// TIA Portal V17 export
// export: Created 2025-03-07T09:19:12.8663943Z, ExportSetting WithDefaults, DisplayName Totally Integrated Automation Portal, DisplayVersion V17 Update 8, DisplayName TIA Portal Openness, DisplayVersion V17 Update 8, DisplayName TIA Portal Version Control Interface, DisplayVersion V17, DisplayName SINAMICS Startdrive Advanced, DisplayVersion V17 SP2, DisplayName SINAMICS Startdrive G110M, G120, G120C, G120D, G120P, G115D, DisplayVersion V17 SP2, DisplayName SINAMICS Startdrive G130, G150, S120, S150, SINAMICS MV, S210, DisplayVersion V17 SP2, DisplayName STEP 7 Professional, DisplayVersion V17 Update 8, DisplayName SINUMERIK ONE STEP 7 Toolbox, DisplayVersion V17 Update 12, DisplayName SINUMERIK 840D sl STEP 7 Toolbox, DisplayVersion V17 Update 12, DisplayName STEP 7 Safety, DisplayVersion V17 Update 6, DisplayName WinCC Advanced, DisplayVersion V17 Update 8
FUNCTION "FC7236_SHOW_HIDE_ELEMENTS_CLADDING" : Void   // FC7236, LAD
{ S7_Optimized_Access := 'FALSE' }
AUTHOR : ETXETAR
VERSION : 1.0
// stored: AutoNumber false, IsIECCheckEnabled false, SetENOAutomatically false, UDAEnableTagReadback false
   VAR_TEMP
      ONE : Byte;
      RETVAL_FILL : Int;
      ZERO : Byte;
      MINUS_ONE : Byte;
      SHOW_TABLES : Bool;
      NO_REASON_CODE : Bool;
      AXIS_AUX1 : Bool;
      AXIS_AUX2 : Bool;
   END_VAR
   VAR_TEMP   // added for the SCL form of the ladder/FBD networks
      _w1 : Bool;
      _w2 : Bool;
   END_VAR
BEGIN

REGION Network 1: MOVE VALUES
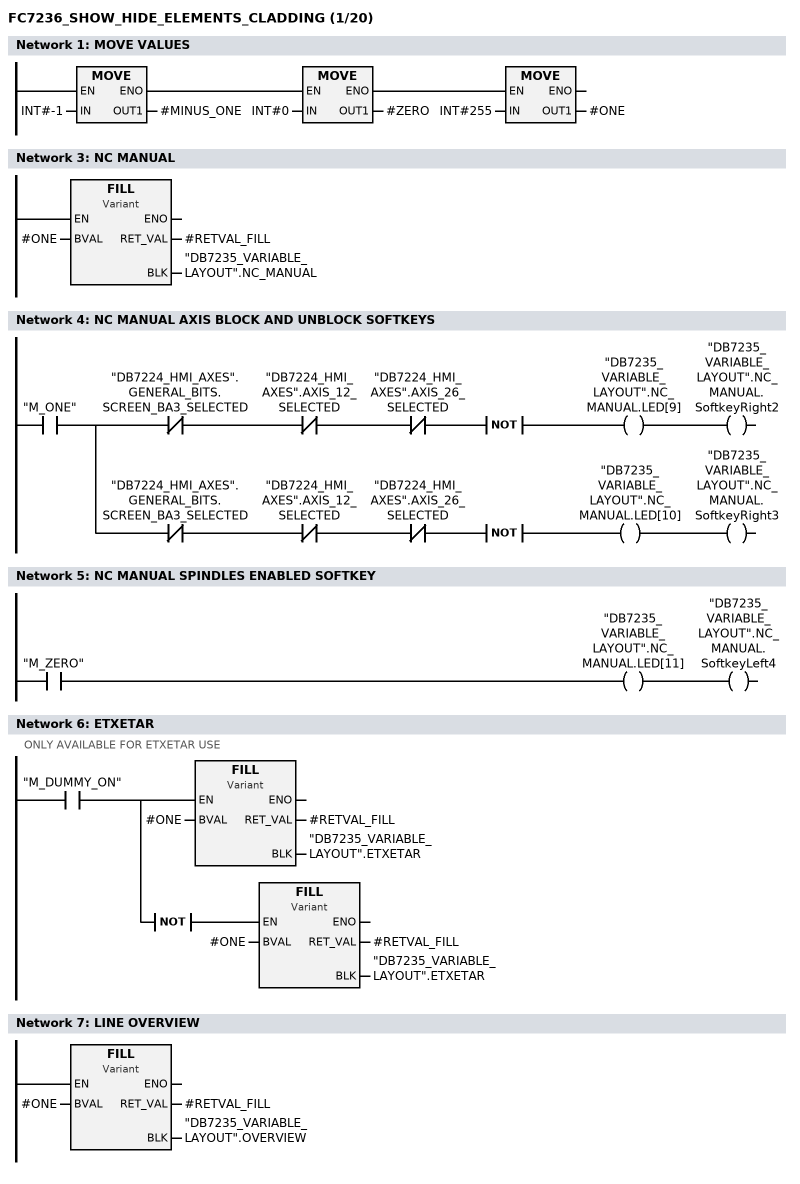
   RUNG wire#powerrail
      { S7_GenerateENO := "TRUE" } Move(in := INT#-1, out1 => #MINUS_ONE)
      { S7_GenerateENO := "TRUE" } Move(in := INT#0, out1 => #ZERO)
      { S7_GenerateENO := "TRUE" } Move(in := INT#255, out1 => #ONE)
   END_RUNG
   // the same network as SCL:
   // ENO of a box is taken as its EN; it also drops when the box reports an error
   #MINUS_ONE := INT#-1;
   #ZERO := INT#0;
   #ONE := INT#255;
END_REGION

REGION Network 2: *************** SHOW OR HIDE ELEMENTS ***************
END_REGION

REGION Network 3: NC MANUAL
   RUNG wire#powerrail
      { S7_Templates := "ptr_type := Variant" } FILL(BVAL := #ONE, RET_VAL => #RETVAL_FILL, BLK => "DB7235_VARIABLE_LAYOUT".NC_MANUAL)
   END_RUNG
   // the same network as SCL:
   #RETVAL_FILL := FILL(BVAL := #ONE, BLK => "DB7235_VARIABLE_LAYOUT".NC_MANUAL);
END_REGION

REGION Network 4: NC MANUAL AXIS BLOCK AND UNBLOCK SOFTKEYS
   RUNG wire#powerrail
      Contact( "M_ONE" )
      wire#w1
      I_Contact( "DB7224_HMI_AXES".GENERAL_BITS.SCREEN_BA3_SELECTED )
      I_Contact( "DB7224_HMI_AXES".AXIS_12_SELECTED )
      I_Contact( "DB7224_HMI_AXES".AXIS_26_SELECTED )
      Not()
      Coil( "DB7235_VARIABLE_LAYOUT".NC_MANUAL.LED[9] )
      Coil( "DB7235_VARIABLE_LAYOUT".NC_MANUAL.SoftkeyRight2 )
   END_RUNG
   RUNG wire#w1
      I_Contact( "DB7224_HMI_AXES".GENERAL_BITS.SCREEN_BA3_SELECTED )
      I_Contact( "DB7224_HMI_AXES".AXIS_12_SELECTED )
      I_Contact( "DB7224_HMI_AXES".AXIS_26_SELECTED )
      Not()
      Coil( "DB7235_VARIABLE_LAYOUT".NC_MANUAL.LED[10] )
      Coil( "DB7235_VARIABLE_LAYOUT".NC_MANUAL.SoftkeyRight3 )
   END_RUNG
   // the same network as SCL:
   "DB7235_VARIABLE_LAYOUT".NC_MANUAL.LED[9] := NOT ("M_ONE" AND NOT "DB7224_HMI_AXES".GENERAL_BITS.SCREEN_BA3_SELECTED AND NOT "DB7224_HMI_AXES".AXIS_12_SELECTED AND NOT "DB7224_HMI_AXES".AXIS_26_SELECTED);
   "DB7235_VARIABLE_LAYOUT".NC_MANUAL.SoftkeyRight2 := NOT ("M_ONE" AND NOT "DB7224_HMI_AXES".GENERAL_BITS.SCREEN_BA3_SELECTED AND NOT "DB7224_HMI_AXES".AXIS_12_SELECTED AND NOT "DB7224_HMI_AXES".AXIS_26_SELECTED);
   "DB7235_VARIABLE_LAYOUT".NC_MANUAL.LED[10] := NOT ("M_ONE" AND NOT "DB7224_HMI_AXES".GENERAL_BITS.SCREEN_BA3_SELECTED AND NOT "DB7224_HMI_AXES".AXIS_12_SELECTED AND NOT "DB7224_HMI_AXES".AXIS_26_SELECTED);
   "DB7235_VARIABLE_LAYOUT".NC_MANUAL.SoftkeyRight3 := NOT ("M_ONE" AND NOT "DB7224_HMI_AXES".GENERAL_BITS.SCREEN_BA3_SELECTED AND NOT "DB7224_HMI_AXES".AXIS_12_SELECTED AND NOT "DB7224_HMI_AXES".AXIS_26_SELECTED);
END_REGION

REGION Network 5: NC MANUAL SPINDLES ENABLED SOFTKEY
   RUNG wire#powerrail
      Contact( "M_ZERO" )
      Coil( "DB7235_VARIABLE_LAYOUT".NC_MANUAL.LED[11] )
      Coil( "DB7235_VARIABLE_LAYOUT".NC_MANUAL.SoftkeyLeft4 )
   END_RUNG
   // the same network as SCL:
   "DB7235_VARIABLE_LAYOUT".NC_MANUAL.LED[11] := "M_ZERO";
   "DB7235_VARIABLE_LAYOUT".NC_MANUAL.SoftkeyLeft4 := "M_ZERO";
END_REGION

REGION Network 6: ETXETAR
   // ONLY AVAILABLE FOR ETXETAR USE
   RUNG wire#powerrail
      Contact( "M_DUMMY_ON" )
      wire#w1
      { S7_Templates := "ptr_type := Variant" } FILL(BVAL := #ONE, RET_VAL => #RETVAL_FILL, BLK => "DB7235_VARIABLE_LAYOUT".ETXETAR)
   END_RUNG
   RUNG wire#w1
      Not()
      { S7_Templates := "ptr_type := Variant" } FILL(BVAL := #ONE, RET_VAL => #RETVAL_FILL, BLK => "DB7235_VARIABLE_LAYOUT".ETXETAR)
   END_RUNG
   // the same network as SCL:
   #_w1 := "M_DUMMY_ON";
   IF #_w1 THEN #RETVAL_FILL := FILL(BVAL := #ONE, BLK => "DB7235_VARIABLE_LAYOUT".ETXETAR); END_IF;
   IF NOT #_w1 THEN #RETVAL_FILL := FILL(BVAL := #ONE, BLK => "DB7235_VARIABLE_LAYOUT".ETXETAR); END_IF;
END_REGION

REGION Network 7: LINE OVERVIEW
   RUNG wire#powerrail
      { S7_Templates := "ptr_type := Variant" } FILL(BVAL := #ONE, RET_VAL => #RETVAL_FILL, BLK => "DB7235_VARIABLE_LAYOUT".OVERVIEW)
   END_RUNG
   // the same network as SCL:
   #RETVAL_FILL := FILL(BVAL := #ONE, BLK => "DB7235_VARIABLE_LAYOUT".OVERVIEW);
END_REGION

REGION Network 8: LINE OVERVIEW IO FIELD AND TEXTS
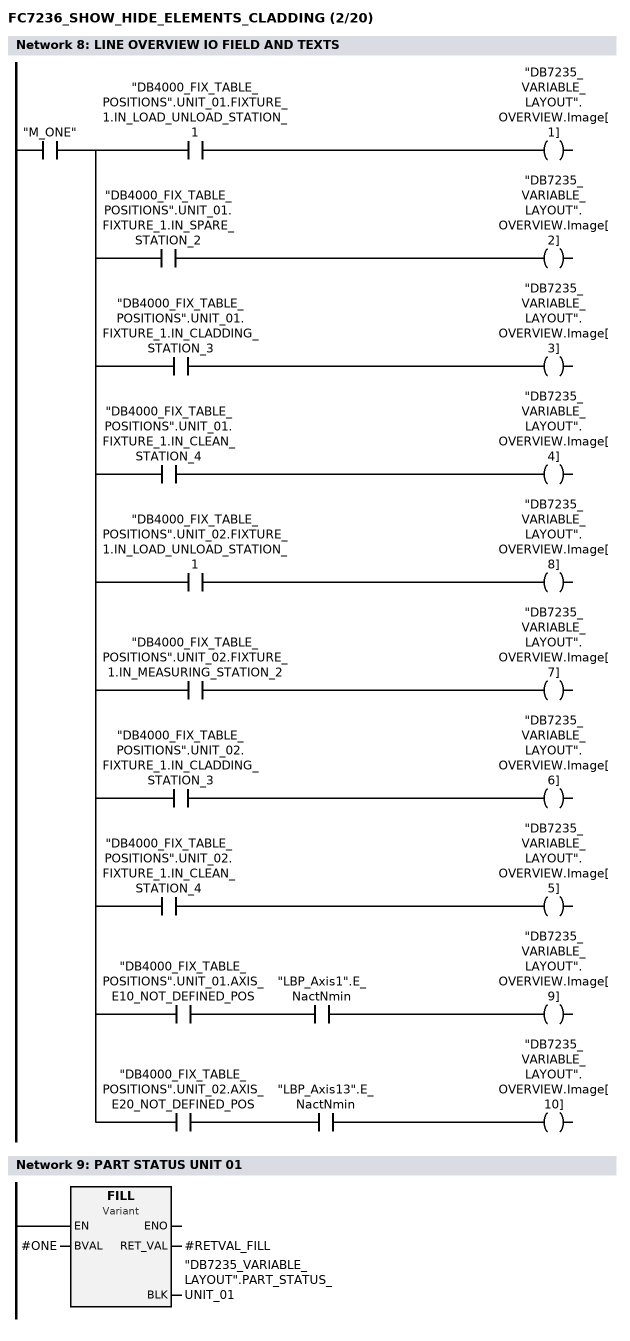
   RUNG wire#powerrail
      Contact( "M_ONE" )
      wire#w1
      Contact( "DB4000_FIX_TABLE_POSITIONS".UNIT_01.FIXTURE_1.IN_LOAD_UNLOAD_STATION_1 )
      Coil( "DB7235_VARIABLE_LAYOUT".OVERVIEW.Image[1] )
   END_RUNG
   RUNG wire#w1
      Contact( "DB4000_FIX_TABLE_POSITIONS".UNIT_01.FIXTURE_1.IN_SPARE_STATION_2 )
      Coil( "DB7235_VARIABLE_LAYOUT".OVERVIEW.Image[2] )
   END_RUNG
   RUNG wire#w1
      Contact( "DB4000_FIX_TABLE_POSITIONS".UNIT_01.FIXTURE_1.IN_CLADDING_STATION_3 )
      Coil( "DB7235_VARIABLE_LAYOUT".OVERVIEW.Image[3] )
   END_RUNG
   RUNG wire#w1
      Contact( "DB4000_FIX_TABLE_POSITIONS".UNIT_01.FIXTURE_1.IN_CLEAN_STATION_4 )
      Coil( "DB7235_VARIABLE_LAYOUT".OVERVIEW.Image[4] )
   END_RUNG
   RUNG wire#w1
      Contact( "DB4000_FIX_TABLE_POSITIONS".UNIT_02.FIXTURE_1.IN_LOAD_UNLOAD_STATION_1 )
      Coil( "DB7235_VARIABLE_LAYOUT".OVERVIEW.Image[8] )
   END_RUNG
   RUNG wire#w1
      Contact( "DB4000_FIX_TABLE_POSITIONS".UNIT_02.FIXTURE_1.IN_MEASURING_STATION_2 )
      Coil( "DB7235_VARIABLE_LAYOUT".OVERVIEW.Image[7] )
   END_RUNG
   RUNG wire#w1
      Contact( "DB4000_FIX_TABLE_POSITIONS".UNIT_02.FIXTURE_1.IN_CLADDING_STATION_3 )
      Coil( "DB7235_VARIABLE_LAYOUT".OVERVIEW.Image[6] )
   END_RUNG
   RUNG wire#w1
      Contact( "DB4000_FIX_TABLE_POSITIONS".UNIT_02.FIXTURE_1.IN_CLEAN_STATION_4 )
      Coil( "DB7235_VARIABLE_LAYOUT".OVERVIEW.Image[5] )
   END_RUNG
   RUNG wire#w1
      Contact( "DB4000_FIX_TABLE_POSITIONS".UNIT_01.AXIS_E10_NOT_DEFINED_POS )
      Contact( "LBP_Axis1".E_NactNmin )
      Coil( "DB7235_VARIABLE_LAYOUT".OVERVIEW.Image[9] )
   END_RUNG
   RUNG wire#w1
      Contact( "DB4000_FIX_TABLE_POSITIONS".UNIT_02.AXIS_E20_NOT_DEFINED_POS )
      Contact( "LBP_Axis13".E_NactNmin )
      Coil( "DB7235_VARIABLE_LAYOUT".OVERVIEW.Image[10] )
   END_RUNG
   // the same network as SCL:
   "DB7235_VARIABLE_LAYOUT".OVERVIEW.Image[1] := "M_ONE" AND "DB4000_FIX_TABLE_POSITIONS".UNIT_01.FIXTURE_1.IN_LOAD_UNLOAD_STATION_1;
   "DB7235_VARIABLE_LAYOUT".OVERVIEW.Image[2] := "M_ONE" AND "DB4000_FIX_TABLE_POSITIONS".UNIT_01.FIXTURE_1.IN_SPARE_STATION_2;
   "DB7235_VARIABLE_LAYOUT".OVERVIEW.Image[3] := "M_ONE" AND "DB4000_FIX_TABLE_POSITIONS".UNIT_01.FIXTURE_1.IN_CLADDING_STATION_3;
   "DB7235_VARIABLE_LAYOUT".OVERVIEW.Image[4] := "M_ONE" AND "DB4000_FIX_TABLE_POSITIONS".UNIT_01.FIXTURE_1.IN_CLEAN_STATION_4;
   "DB7235_VARIABLE_LAYOUT".OVERVIEW.Image[8] := "M_ONE" AND "DB4000_FIX_TABLE_POSITIONS".UNIT_02.FIXTURE_1.IN_LOAD_UNLOAD_STATION_1;
   "DB7235_VARIABLE_LAYOUT".OVERVIEW.Image[7] := "M_ONE" AND "DB4000_FIX_TABLE_POSITIONS".UNIT_02.FIXTURE_1.IN_MEASURING_STATION_2;
   "DB7235_VARIABLE_LAYOUT".OVERVIEW.Image[6] := "M_ONE" AND "DB4000_FIX_TABLE_POSITIONS".UNIT_02.FIXTURE_1.IN_CLADDING_STATION_3;
   "DB7235_VARIABLE_LAYOUT".OVERVIEW.Image[5] := "M_ONE" AND "DB4000_FIX_TABLE_POSITIONS".UNIT_02.FIXTURE_1.IN_CLEAN_STATION_4;
   "DB7235_VARIABLE_LAYOUT".OVERVIEW.Image[9] := "M_ONE" AND "DB4000_FIX_TABLE_POSITIONS".UNIT_01.AXIS_E10_NOT_DEFINED_POS AND "LBP_Axis1".E_NactNmin;
   "DB7235_VARIABLE_LAYOUT".OVERVIEW.Image[10] := "M_ONE" AND "DB4000_FIX_TABLE_POSITIONS".UNIT_02.AXIS_E20_NOT_DEFINED_POS AND "LBP_Axis13".E_NactNmin;
END_REGION

REGION Network 9: PART STATUS UNIT 01
   RUNG wire#powerrail
      { S7_Templates := "ptr_type := Variant" } FILL(BVAL := #ONE, RET_VAL => #RETVAL_FILL, BLK => "DB7235_VARIABLE_LAYOUT".PART_STATUS_UNIT_01)
   END_RUNG
   // the same network as SCL:
   #RETVAL_FILL := FILL(BVAL := #ONE, BLK => "DB7235_VARIABLE_LAYOUT".PART_STATUS_UNIT_01);
END_REGION

REGION Network 10: PART STATUS IO FIELD AND TEXTS UNIT 01
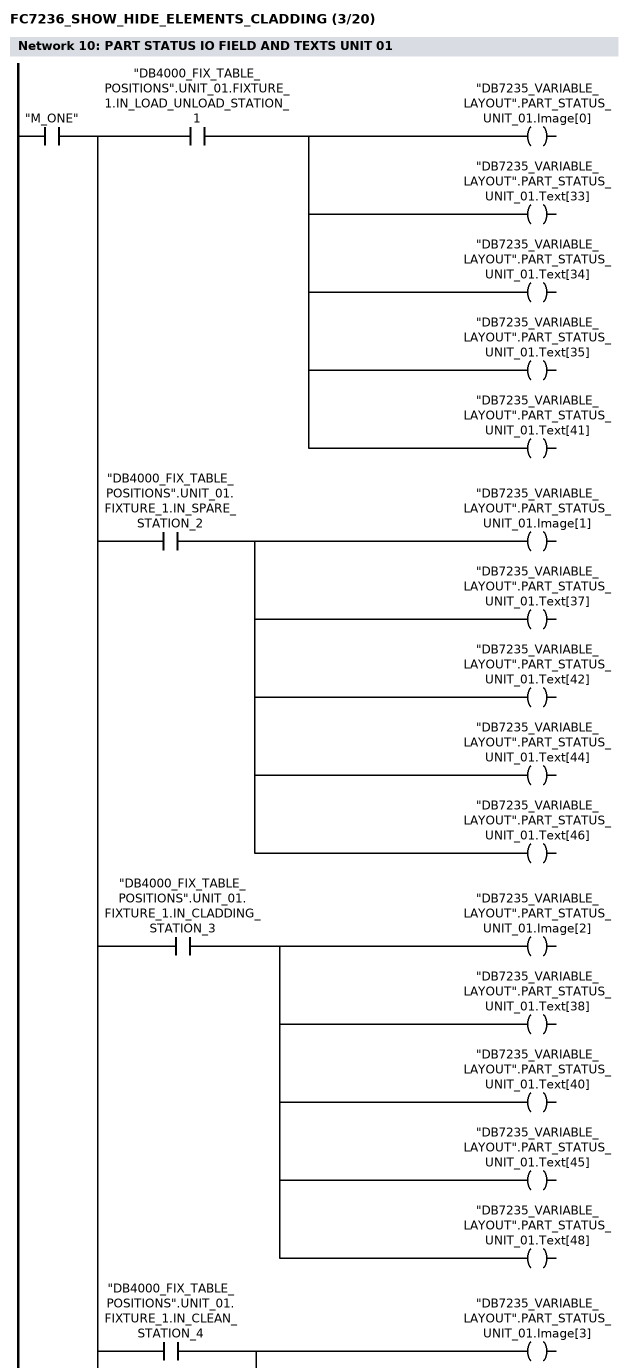
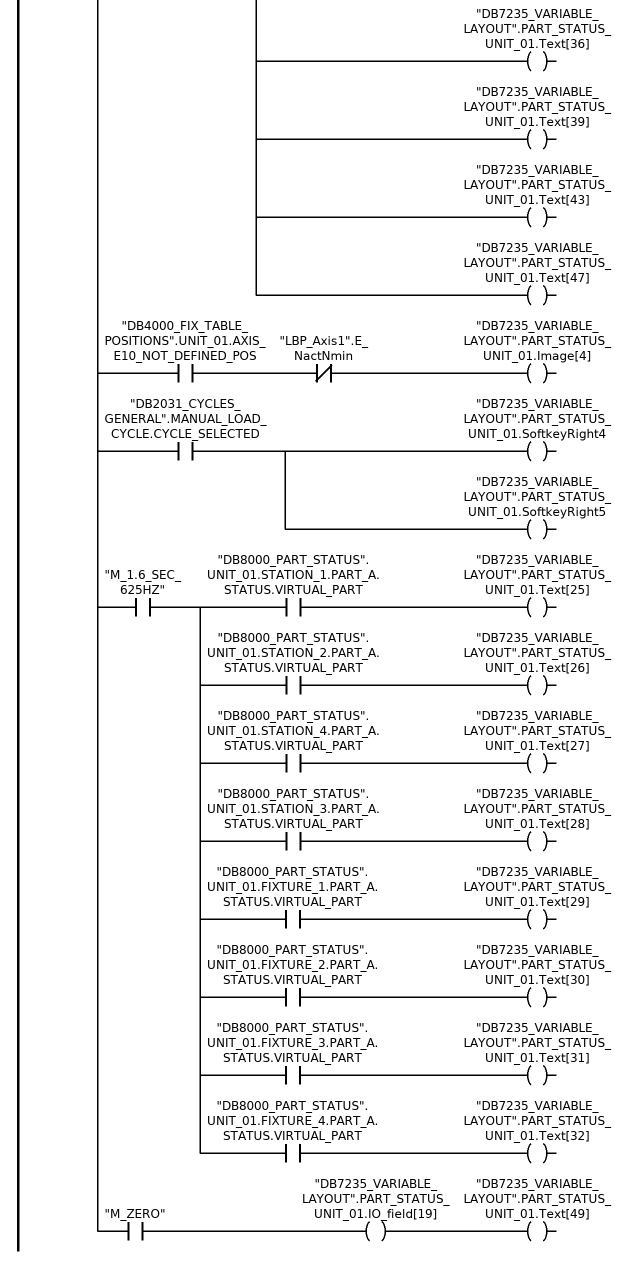
   RUNG wire#powerrail
      Contact( "M_ONE" )
      wire#w1
      Contact( "DB4000_FIX_TABLE_POSITIONS".UNIT_01.FIXTURE_1.IN_LOAD_UNLOAD_STATION_1 )
      wire#w2
      Coil( "DB7235_VARIABLE_LAYOUT".PART_STATUS_UNIT_01.Image[0] )
   END_RUNG
   RUNG wire#w2
      Coil( "DB7235_VARIABLE_LAYOUT".PART_STATUS_UNIT_01.Text[33] )
   END_RUNG
   RUNG wire#w2
      Coil( "DB7235_VARIABLE_LAYOUT".PART_STATUS_UNIT_01.Text[34] )
   END_RUNG
   RUNG wire#w2
      Coil( "DB7235_VARIABLE_LAYOUT".PART_STATUS_UNIT_01.Text[35] )
   END_RUNG
   RUNG wire#w2
      Coil( "DB7235_VARIABLE_LAYOUT".PART_STATUS_UNIT_01.Text[41] )
   END_RUNG
   RUNG wire#w1
      Contact( "DB4000_FIX_TABLE_POSITIONS".UNIT_01.FIXTURE_1.IN_SPARE_STATION_2 )
      wire#w3
      Coil( "DB7235_VARIABLE_LAYOUT".PART_STATUS_UNIT_01.Image[1] )
   END_RUNG
   RUNG wire#w3
      Coil( "DB7235_VARIABLE_LAYOUT".PART_STATUS_UNIT_01.Text[37] )
   END_RUNG
   RUNG wire#w3
      Coil( "DB7235_VARIABLE_LAYOUT".PART_STATUS_UNIT_01.Text[42] )
   END_RUNG
   RUNG wire#w3
      Coil( "DB7235_VARIABLE_LAYOUT".PART_STATUS_UNIT_01.Text[44] )
   END_RUNG
   RUNG wire#w3
      Coil( "DB7235_VARIABLE_LAYOUT".PART_STATUS_UNIT_01.Text[46] )
   END_RUNG
   RUNG wire#w1
      Contact( "DB4000_FIX_TABLE_POSITIONS".UNIT_01.FIXTURE_1.IN_CLADDING_STATION_3 )
      wire#w4
      Coil( "DB7235_VARIABLE_LAYOUT".PART_STATUS_UNIT_01.Image[2] )
   END_RUNG
   RUNG wire#w4
      Coil( "DB7235_VARIABLE_LAYOUT".PART_STATUS_UNIT_01.Text[38] )
   END_RUNG
   RUNG wire#w4
      Coil( "DB7235_VARIABLE_LAYOUT".PART_STATUS_UNIT_01.Text[40] )
   END_RUNG
   RUNG wire#w4
      Coil( "DB7235_VARIABLE_LAYOUT".PART_STATUS_UNIT_01.Text[45] )
   END_RUNG
   RUNG wire#w4
      Coil( "DB7235_VARIABLE_LAYOUT".PART_STATUS_UNIT_01.Text[48] )
   END_RUNG
   RUNG wire#w1
      Contact( "DB4000_FIX_TABLE_POSITIONS".UNIT_01.FIXTURE_1.IN_CLEAN_STATION_4 )
      wire#w5
      Coil( "DB7235_VARIABLE_LAYOUT".PART_STATUS_UNIT_01.Image[3] )
   END_RUNG
   RUNG wire#w5
      Coil( "DB7235_VARIABLE_LAYOUT".PART_STATUS_UNIT_01.Text[36] )
   END_RUNG
   RUNG wire#w5
      Coil( "DB7235_VARIABLE_LAYOUT".PART_STATUS_UNIT_01.Text[39] )
   END_RUNG
   RUNG wire#w5
      Coil( "DB7235_VARIABLE_LAYOUT".PART_STATUS_UNIT_01.Text[43] )
   END_RUNG
   RUNG wire#w5
      Coil( "DB7235_VARIABLE_LAYOUT".PART_STATUS_UNIT_01.Text[47] )
   END_RUNG
   RUNG wire#w1
      Contact( "DB4000_FIX_TABLE_POSITIONS".UNIT_01.AXIS_E10_NOT_DEFINED_POS )
      I_Contact( "LBP_Axis1".E_NactNmin )
      Coil( "DB7235_VARIABLE_LAYOUT".PART_STATUS_UNIT_01.Image[4] )
   END_RUNG
   RUNG wire#w1
      Contact( "DB2031_CYCLES_GENERAL".MANUAL_LOAD_CYCLE.CYCLE_SELECTED )
      wire#w6
      Coil( "DB7235_VARIABLE_LAYOUT".PART_STATUS_UNIT_01.SoftkeyRight4 )
   END_RUNG
   RUNG wire#w6
      Coil( "DB7235_VARIABLE_LAYOUT".PART_STATUS_UNIT_01.SoftkeyRight5 )
   END_RUNG
   RUNG wire#w1
      Contact( "M_1.6_SEC_625HZ" )
      wire#w7
      Contact( "DB8000_PART_STATUS".UNIT_01.STATION_1.PART_A.STATUS.VIRTUAL_PART )
      Coil( "DB7235_VARIABLE_LAYOUT".PART_STATUS_UNIT_01.Text[25] )
   END_RUNG
   RUNG wire#w7
      Contact( "DB8000_PART_STATUS".UNIT_01.STATION_2.PART_A.STATUS.VIRTUAL_PART )
      Coil( "DB7235_VARIABLE_LAYOUT".PART_STATUS_UNIT_01.Text[26] )
   END_RUNG
   RUNG wire#w7
      Contact( "DB8000_PART_STATUS".UNIT_01.STATION_4.PART_A.STATUS.VIRTUAL_PART )
      Coil( "DB7235_VARIABLE_LAYOUT".PART_STATUS_UNIT_01.Text[27] )
   END_RUNG
   RUNG wire#w7
      Contact( "DB8000_PART_STATUS".UNIT_01.STATION_3.PART_A.STATUS.VIRTUAL_PART )
      Coil( "DB7235_VARIABLE_LAYOUT".PART_STATUS_UNIT_01.Text[28] )
   END_RUNG
   RUNG wire#w7
      Contact( "DB8000_PART_STATUS".UNIT_01.FIXTURE_1.PART_A.STATUS.VIRTUAL_PART )
      Coil( "DB7235_VARIABLE_LAYOUT".PART_STATUS_UNIT_01.Text[29] )
   END_RUNG
   RUNG wire#w7
      Contact( "DB8000_PART_STATUS".UNIT_01.FIXTURE_2.PART_A.STATUS.VIRTUAL_PART )
      Coil( "DB7235_VARIABLE_LAYOUT".PART_STATUS_UNIT_01.Text[30] )
   END_RUNG
   RUNG wire#w7
      Contact( "DB8000_PART_STATUS".UNIT_01.FIXTURE_3.PART_A.STATUS.VIRTUAL_PART )
      Coil( "DB7235_VARIABLE_LAYOUT".PART_STATUS_UNIT_01.Text[31] )
   END_RUNG
   RUNG wire#w7
      Contact( "DB8000_PART_STATUS".UNIT_01.FIXTURE_4.PART_A.STATUS.VIRTUAL_PART )
      Coil( "DB7235_VARIABLE_LAYOUT".PART_STATUS_UNIT_01.Text[32] )
   END_RUNG
   RUNG wire#w1
      Contact( "M_ZERO" )
      Coil( "DB7235_VARIABLE_LAYOUT".PART_STATUS_UNIT_01.IO_field[19] )
      Coil( "DB7235_VARIABLE_LAYOUT".PART_STATUS_UNIT_01.Text[49] )
   END_RUNG
   // the same network as SCL:
   "DB7235_VARIABLE_LAYOUT".PART_STATUS_UNIT_01.Image[0] := "M_ONE" AND "DB4000_FIX_TABLE_POSITIONS".UNIT_01.FIXTURE_1.IN_LOAD_UNLOAD_STATION_1;
   "DB7235_VARIABLE_LAYOUT".PART_STATUS_UNIT_01.Text[33] := "M_ONE" AND "DB4000_FIX_TABLE_POSITIONS".UNIT_01.FIXTURE_1.IN_LOAD_UNLOAD_STATION_1;
   "DB7235_VARIABLE_LAYOUT".PART_STATUS_UNIT_01.Text[34] := "M_ONE" AND "DB4000_FIX_TABLE_POSITIONS".UNIT_01.FIXTURE_1.IN_LOAD_UNLOAD_STATION_1;
   "DB7235_VARIABLE_LAYOUT".PART_STATUS_UNIT_01.Text[35] := "M_ONE" AND "DB4000_FIX_TABLE_POSITIONS".UNIT_01.FIXTURE_1.IN_LOAD_UNLOAD_STATION_1;
   "DB7235_VARIABLE_LAYOUT".PART_STATUS_UNIT_01.Text[41] := "M_ONE" AND "DB4000_FIX_TABLE_POSITIONS".UNIT_01.FIXTURE_1.IN_LOAD_UNLOAD_STATION_1;
   "DB7235_VARIABLE_LAYOUT".PART_STATUS_UNIT_01.Image[1] := "M_ONE" AND "DB4000_FIX_TABLE_POSITIONS".UNIT_01.FIXTURE_1.IN_SPARE_STATION_2;
   "DB7235_VARIABLE_LAYOUT".PART_STATUS_UNIT_01.Text[37] := "M_ONE" AND "DB4000_FIX_TABLE_POSITIONS".UNIT_01.FIXTURE_1.IN_SPARE_STATION_2;
   "DB7235_VARIABLE_LAYOUT".PART_STATUS_UNIT_01.Text[42] := "M_ONE" AND "DB4000_FIX_TABLE_POSITIONS".UNIT_01.FIXTURE_1.IN_SPARE_STATION_2;
   "DB7235_VARIABLE_LAYOUT".PART_STATUS_UNIT_01.Text[44] := "M_ONE" AND "DB4000_FIX_TABLE_POSITIONS".UNIT_01.FIXTURE_1.IN_SPARE_STATION_2;
   "DB7235_VARIABLE_LAYOUT".PART_STATUS_UNIT_01.Text[46] := "M_ONE" AND "DB4000_FIX_TABLE_POSITIONS".UNIT_01.FIXTURE_1.IN_SPARE_STATION_2;
   "DB7235_VARIABLE_LAYOUT".PART_STATUS_UNIT_01.Image[2] := "M_ONE" AND "DB4000_FIX_TABLE_POSITIONS".UNIT_01.FIXTURE_1.IN_CLADDING_STATION_3;
   "DB7235_VARIABLE_LAYOUT".PART_STATUS_UNIT_01.Text[38] := "M_ONE" AND "DB4000_FIX_TABLE_POSITIONS".UNIT_01.FIXTURE_1.IN_CLADDING_STATION_3;
   "DB7235_VARIABLE_LAYOUT".PART_STATUS_UNIT_01.Text[40] := "M_ONE" AND "DB4000_FIX_TABLE_POSITIONS".UNIT_01.FIXTURE_1.IN_CLADDING_STATION_3;
   "DB7235_VARIABLE_LAYOUT".PART_STATUS_UNIT_01.Text[45] := "M_ONE" AND "DB4000_FIX_TABLE_POSITIONS".UNIT_01.FIXTURE_1.IN_CLADDING_STATION_3;
   "DB7235_VARIABLE_LAYOUT".PART_STATUS_UNIT_01.Text[48] := "M_ONE" AND "DB4000_FIX_TABLE_POSITIONS".UNIT_01.FIXTURE_1.IN_CLADDING_STATION_3;
   "DB7235_VARIABLE_LAYOUT".PART_STATUS_UNIT_01.Image[3] := "M_ONE" AND "DB4000_FIX_TABLE_POSITIONS".UNIT_01.FIXTURE_1.IN_CLEAN_STATION_4;
   "DB7235_VARIABLE_LAYOUT".PART_STATUS_UNIT_01.Text[36] := "M_ONE" AND "DB4000_FIX_TABLE_POSITIONS".UNIT_01.FIXTURE_1.IN_CLEAN_STATION_4;
   "DB7235_VARIABLE_LAYOUT".PART_STATUS_UNIT_01.Text[39] := "M_ONE" AND "DB4000_FIX_TABLE_POSITIONS".UNIT_01.FIXTURE_1.IN_CLEAN_STATION_4;
   "DB7235_VARIABLE_LAYOUT".PART_STATUS_UNIT_01.Text[43] := "M_ONE" AND "DB4000_FIX_TABLE_POSITIONS".UNIT_01.FIXTURE_1.IN_CLEAN_STATION_4;
   "DB7235_VARIABLE_LAYOUT".PART_STATUS_UNIT_01.Text[47] := "M_ONE" AND "DB4000_FIX_TABLE_POSITIONS".UNIT_01.FIXTURE_1.IN_CLEAN_STATION_4;
   "DB7235_VARIABLE_LAYOUT".PART_STATUS_UNIT_01.Image[4] := "M_ONE" AND "DB4000_FIX_TABLE_POSITIONS".UNIT_01.AXIS_E10_NOT_DEFINED_POS AND NOT "LBP_Axis1".E_NactNmin;
   "DB7235_VARIABLE_LAYOUT".PART_STATUS_UNIT_01.SoftkeyRight4 := "M_ONE" AND "DB2031_CYCLES_GENERAL".MANUAL_LOAD_CYCLE.CYCLE_SELECTED;
   "DB7235_VARIABLE_LAYOUT".PART_STATUS_UNIT_01.SoftkeyRight5 := "DB7235_VARIABLE_LAYOUT".PART_STATUS_UNIT_01.SoftkeyRight4;
   #_w1 := "M_ONE" AND "M_1.6_SEC_625HZ";
   "DB7235_VARIABLE_LAYOUT".PART_STATUS_UNIT_01.Text[25] := #_w1 AND "DB8000_PART_STATUS".UNIT_01.STATION_1.PART_A.STATUS.VIRTUAL_PART;
   "DB7235_VARIABLE_LAYOUT".PART_STATUS_UNIT_01.Text[26] := #_w1 AND "DB8000_PART_STATUS".UNIT_01.STATION_2.PART_A.STATUS.VIRTUAL_PART;
   "DB7235_VARIABLE_LAYOUT".PART_STATUS_UNIT_01.Text[27] := #_w1 AND "DB8000_PART_STATUS".UNIT_01.STATION_4.PART_A.STATUS.VIRTUAL_PART;
   "DB7235_VARIABLE_LAYOUT".PART_STATUS_UNIT_01.Text[28] := #_w1 AND "DB8000_PART_STATUS".UNIT_01.STATION_3.PART_A.STATUS.VIRTUAL_PART;
   "DB7235_VARIABLE_LAYOUT".PART_STATUS_UNIT_01.Text[29] := #_w1 AND "DB8000_PART_STATUS".UNIT_01.FIXTURE_1.PART_A.STATUS.VIRTUAL_PART;
   "DB7235_VARIABLE_LAYOUT".PART_STATUS_UNIT_01.Text[30] := #_w1 AND "DB8000_PART_STATUS".UNIT_01.FIXTURE_2.PART_A.STATUS.VIRTUAL_PART;
   "DB7235_VARIABLE_LAYOUT".PART_STATUS_UNIT_01.Text[31] := #_w1 AND "DB8000_PART_STATUS".UNIT_01.FIXTURE_3.PART_A.STATUS.VIRTUAL_PART;
   "DB7235_VARIABLE_LAYOUT".PART_STATUS_UNIT_01.Text[32] := #_w1 AND "DB8000_PART_STATUS".UNIT_01.FIXTURE_4.PART_A.STATUS.VIRTUAL_PART;
   "DB7235_VARIABLE_LAYOUT".PART_STATUS_UNIT_01.IO_field[19] := "M_ONE" AND "M_ZERO";
   "DB7235_VARIABLE_LAYOUT".PART_STATUS_UNIT_01.Text[49] := "M_ONE" AND "M_ZERO";
END_REGION

REGION Network 11: QUALITY CHECK
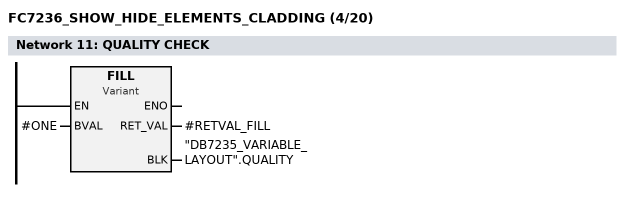
   RUNG wire#powerrail
      { S7_Templates := "ptr_type := Variant" } FILL(BVAL := #ONE, RET_VAL => #RETVAL_FILL, BLK => "DB7235_VARIABLE_LAYOUT".QUALITY)
   END_RUNG
   // the same network as SCL:
   #RETVAL_FILL := FILL(BVAL := #ONE, BLK => "DB7235_VARIABLE_LAYOUT".QUALITY);
END_REGION

REGION Network 12: QUALITY CHECK IO FIELD AND TEXTS
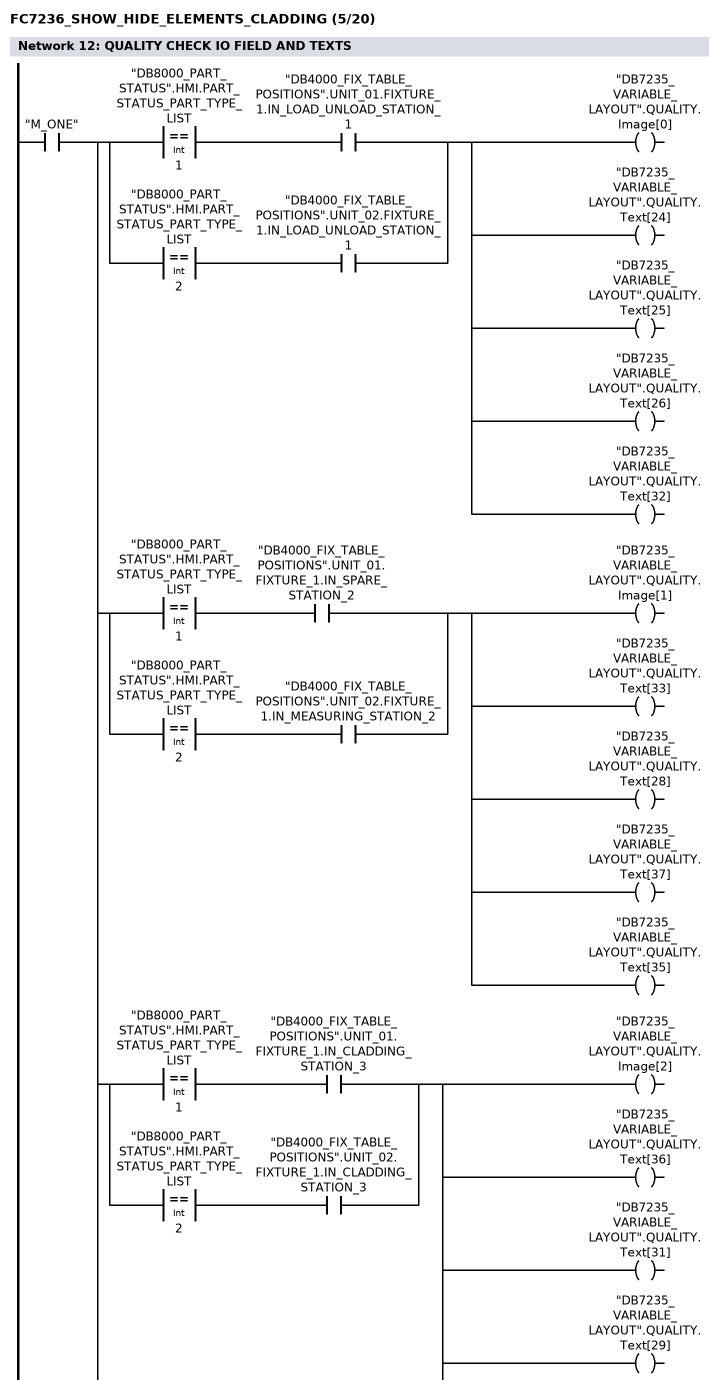
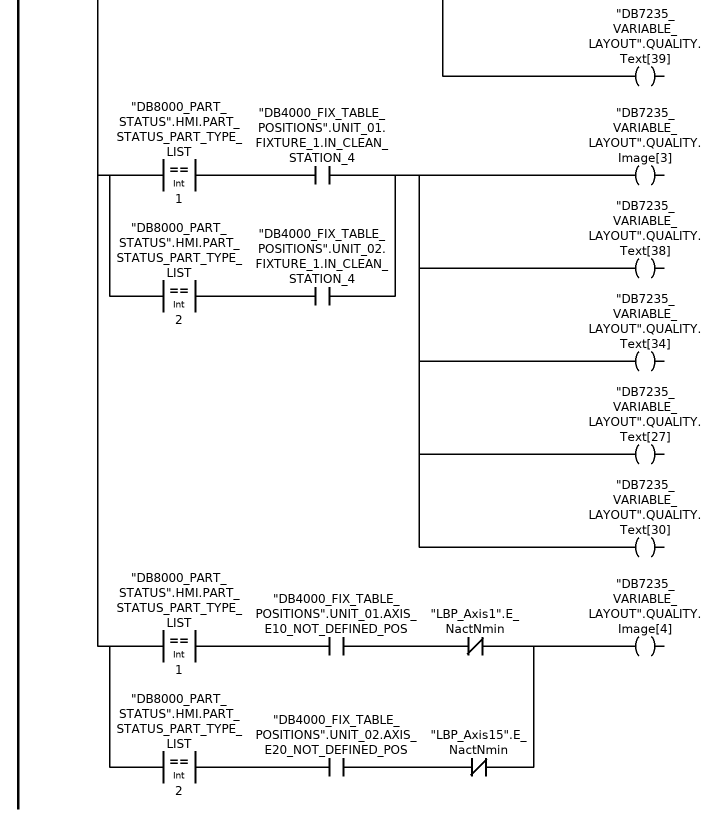
   RUNG wire#powerrail
      Contact( "M_ONE" )
      wire#w1
      { S7_Templates := "SrcType := Int" } EQ_Contact(in1 := "DB8000_PART_STATUS".HMI.PART_STATUS_PART_TYPE_LIST, in2 := 1)
      Contact( "DB4000_FIX_TABLE_POSITIONS".UNIT_01.FIXTURE_1.IN_LOAD_UNLOAD_STATION_1 )
      wire#w2
      Coil( "DB7235_VARIABLE_LAYOUT".QUALITY.Image[0] )
   END_RUNG
   RUNG wire#w1
      { S7_Templates := "SrcType := Int" } EQ_Contact(in1 := "DB8000_PART_STATUS".HMI.PART_STATUS_PART_TYPE_LIST, in2 := 2)
      Contact( "DB4000_FIX_TABLE_POSITIONS".UNIT_02.FIXTURE_1.IN_LOAD_UNLOAD_STATION_1 )
   END_RUNG wire#w2
   RUNG wire#w2
      Coil( "DB7235_VARIABLE_LAYOUT".QUALITY.Text[24] )
   END_RUNG
   RUNG wire#w2
      Coil( "DB7235_VARIABLE_LAYOUT".QUALITY.Text[25] )
   END_RUNG
   RUNG wire#w2
      Coil( "DB7235_VARIABLE_LAYOUT".QUALITY.Text[26] )
   END_RUNG
   RUNG wire#w2
      Coil( "DB7235_VARIABLE_LAYOUT".QUALITY.Text[32] )
   END_RUNG
   RUNG wire#w1
      { S7_Templates := "SrcType := Int" } EQ_Contact(in1 := "DB8000_PART_STATUS".HMI.PART_STATUS_PART_TYPE_LIST, in2 := 1)
      Contact( "DB4000_FIX_TABLE_POSITIONS".UNIT_01.FIXTURE_1.IN_SPARE_STATION_2 )
      wire#w3
      Coil( "DB7235_VARIABLE_LAYOUT".QUALITY.Image[1] )
   END_RUNG
   RUNG wire#w1
      { S7_Templates := "SrcType := Int" } EQ_Contact(in1 := "DB8000_PART_STATUS".HMI.PART_STATUS_PART_TYPE_LIST, in2 := 2)
      Contact( "DB4000_FIX_TABLE_POSITIONS".UNIT_02.FIXTURE_1.IN_MEASURING_STATION_2 )
   END_RUNG wire#w3
   RUNG wire#w3
      Coil( "DB7235_VARIABLE_LAYOUT".QUALITY.Text[33] )
   END_RUNG
   RUNG wire#w3
      Coil( "DB7235_VARIABLE_LAYOUT".QUALITY.Text[28] )
   END_RUNG
   RUNG wire#w3
      Coil( "DB7235_VARIABLE_LAYOUT".QUALITY.Text[37] )
   END_RUNG
   RUNG wire#w3
      Coil( "DB7235_VARIABLE_LAYOUT".QUALITY.Text[35] )
   END_RUNG
   RUNG wire#w1
      { S7_Templates := "SrcType := Int" } EQ_Contact(in1 := "DB8000_PART_STATUS".HMI.PART_STATUS_PART_TYPE_LIST, in2 := 1)
      Contact( "DB4000_FIX_TABLE_POSITIONS".UNIT_01.FIXTURE_1.IN_CLADDING_STATION_3 )
      wire#w4
      Coil( "DB7235_VARIABLE_LAYOUT".QUALITY.Image[2] )
   END_RUNG
   RUNG wire#w1
      { S7_Templates := "SrcType := Int" } EQ_Contact(in1 := "DB8000_PART_STATUS".HMI.PART_STATUS_PART_TYPE_LIST, in2 := 2)
      Contact( "DB4000_FIX_TABLE_POSITIONS".UNIT_02.FIXTURE_1.IN_CLADDING_STATION_3 )
   END_RUNG wire#w4
   RUNG wire#w4
      Coil( "DB7235_VARIABLE_LAYOUT".QUALITY.Text[36] )
   END_RUNG
   RUNG wire#w4
      Coil( "DB7235_VARIABLE_LAYOUT".QUALITY.Text[31] )
   END_RUNG
   RUNG wire#w4
      Coil( "DB7235_VARIABLE_LAYOUT".QUALITY.Text[29] )
   END_RUNG
   RUNG wire#w4
      Coil( "DB7235_VARIABLE_LAYOUT".QUALITY.Text[39] )
   END_RUNG
   RUNG wire#w1
      { S7_Templates := "SrcType := Int" } EQ_Contact(in1 := "DB8000_PART_STATUS".HMI.PART_STATUS_PART_TYPE_LIST, in2 := 1)
      Contact( "DB4000_FIX_TABLE_POSITIONS".UNIT_01.FIXTURE_1.IN_CLEAN_STATION_4 )
      wire#w5
      Coil( "DB7235_VARIABLE_LAYOUT".QUALITY.Image[3] )
   END_RUNG
   RUNG wire#w1
      { S7_Templates := "SrcType := Int" } EQ_Contact(in1 := "DB8000_PART_STATUS".HMI.PART_STATUS_PART_TYPE_LIST, in2 := 2)
      Contact( "DB4000_FIX_TABLE_POSITIONS".UNIT_02.FIXTURE_1.IN_CLEAN_STATION_4 )
   END_RUNG wire#w5
   RUNG wire#w5
      Coil( "DB7235_VARIABLE_LAYOUT".QUALITY.Text[38] )
   END_RUNG
   RUNG wire#w5
      Coil( "DB7235_VARIABLE_LAYOUT".QUALITY.Text[34] )
   END_RUNG
   RUNG wire#w5
      Coil( "DB7235_VARIABLE_LAYOUT".QUALITY.Text[27] )
   END_RUNG
   RUNG wire#w5
      Coil( "DB7235_VARIABLE_LAYOUT".QUALITY.Text[30] )
   END_RUNG
   RUNG wire#w1
      { S7_Templates := "SrcType := Int" } EQ_Contact(in1 := "DB8000_PART_STATUS".HMI.PART_STATUS_PART_TYPE_LIST, in2 := 1)
      Contact( "DB4000_FIX_TABLE_POSITIONS".UNIT_01.AXIS_E10_NOT_DEFINED_POS )
      I_Contact( "LBP_Axis1".E_NactNmin )
      wire#w6
      Coil( "DB7235_VARIABLE_LAYOUT".QUALITY.Image[4] )
   END_RUNG
   RUNG wire#w1
      { S7_Templates := "SrcType := Int" } EQ_Contact(in1 := "DB8000_PART_STATUS".HMI.PART_STATUS_PART_TYPE_LIST, in2 := 2)
      Contact( "DB4000_FIX_TABLE_POSITIONS".UNIT_02.AXIS_E20_NOT_DEFINED_POS )
      I_Contact( "LBP_Axis15".E_NactNmin )
   END_RUNG wire#w6
   // the same network as SCL:
   "DB7235_VARIABLE_LAYOUT".QUALITY.Image[0] := "M_ONE" AND ((("DB8000_PART_STATUS".HMI.PART_STATUS_PART_TYPE_LIST = 1) AND "DB4000_FIX_TABLE_POSITIONS".UNIT_01.FIXTURE_1.IN_LOAD_UNLOAD_STATION_1) OR (("DB8000_PART_STATUS".HMI.PART_STATUS_PART_TYPE_LIST = 2) AND "DB4000_FIX_TABLE_POSITIONS".UNIT_02.FIXTURE_1.IN_LOAD_UNLOAD_STATION_1));
   "DB7235_VARIABLE_LAYOUT".QUALITY.Text[24] := "M_ONE" AND ((("DB8000_PART_STATUS".HMI.PART_STATUS_PART_TYPE_LIST = 1) AND "DB4000_FIX_TABLE_POSITIONS".UNIT_01.FIXTURE_1.IN_LOAD_UNLOAD_STATION_1) OR (("DB8000_PART_STATUS".HMI.PART_STATUS_PART_TYPE_LIST = 2) AND "DB4000_FIX_TABLE_POSITIONS".UNIT_02.FIXTURE_1.IN_LOAD_UNLOAD_STATION_1));
   "DB7235_VARIABLE_LAYOUT".QUALITY.Text[25] := "M_ONE" AND ((("DB8000_PART_STATUS".HMI.PART_STATUS_PART_TYPE_LIST = 1) AND "DB4000_FIX_TABLE_POSITIONS".UNIT_01.FIXTURE_1.IN_LOAD_UNLOAD_STATION_1) OR (("DB8000_PART_STATUS".HMI.PART_STATUS_PART_TYPE_LIST = 2) AND "DB4000_FIX_TABLE_POSITIONS".UNIT_02.FIXTURE_1.IN_LOAD_UNLOAD_STATION_1));
   "DB7235_VARIABLE_LAYOUT".QUALITY.Text[26] := "M_ONE" AND ((("DB8000_PART_STATUS".HMI.PART_STATUS_PART_TYPE_LIST = 1) AND "DB4000_FIX_TABLE_POSITIONS".UNIT_01.FIXTURE_1.IN_LOAD_UNLOAD_STATION_1) OR (("DB8000_PART_STATUS".HMI.PART_STATUS_PART_TYPE_LIST = 2) AND "DB4000_FIX_TABLE_POSITIONS".UNIT_02.FIXTURE_1.IN_LOAD_UNLOAD_STATION_1));
   "DB7235_VARIABLE_LAYOUT".QUALITY.Text[32] := "M_ONE" AND ((("DB8000_PART_STATUS".HMI.PART_STATUS_PART_TYPE_LIST = 1) AND "DB4000_FIX_TABLE_POSITIONS".UNIT_01.FIXTURE_1.IN_LOAD_UNLOAD_STATION_1) OR (("DB8000_PART_STATUS".HMI.PART_STATUS_PART_TYPE_LIST = 2) AND "DB4000_FIX_TABLE_POSITIONS".UNIT_02.FIXTURE_1.IN_LOAD_UNLOAD_STATION_1));
   "DB7235_VARIABLE_LAYOUT".QUALITY.Image[1] := "M_ONE" AND ((("DB8000_PART_STATUS".HMI.PART_STATUS_PART_TYPE_LIST = 1) AND "DB4000_FIX_TABLE_POSITIONS".UNIT_01.FIXTURE_1.IN_SPARE_STATION_2) OR (("DB8000_PART_STATUS".HMI.PART_STATUS_PART_TYPE_LIST = 2) AND "DB4000_FIX_TABLE_POSITIONS".UNIT_02.FIXTURE_1.IN_MEASURING_STATION_2));
   "DB7235_VARIABLE_LAYOUT".QUALITY.Text[33] := "M_ONE" AND ((("DB8000_PART_STATUS".HMI.PART_STATUS_PART_TYPE_LIST = 1) AND "DB4000_FIX_TABLE_POSITIONS".UNIT_01.FIXTURE_1.IN_SPARE_STATION_2) OR (("DB8000_PART_STATUS".HMI.PART_STATUS_PART_TYPE_LIST = 2) AND "DB4000_FIX_TABLE_POSITIONS".UNIT_02.FIXTURE_1.IN_MEASURING_STATION_2));
   "DB7235_VARIABLE_LAYOUT".QUALITY.Text[28] := "M_ONE" AND ((("DB8000_PART_STATUS".HMI.PART_STATUS_PART_TYPE_LIST = 1) AND "DB4000_FIX_TABLE_POSITIONS".UNIT_01.FIXTURE_1.IN_SPARE_STATION_2) OR (("DB8000_PART_STATUS".HMI.PART_STATUS_PART_TYPE_LIST = 2) AND "DB4000_FIX_TABLE_POSITIONS".UNIT_02.FIXTURE_1.IN_MEASURING_STATION_2));
   "DB7235_VARIABLE_LAYOUT".QUALITY.Text[37] := "M_ONE" AND ((("DB8000_PART_STATUS".HMI.PART_STATUS_PART_TYPE_LIST = 1) AND "DB4000_FIX_TABLE_POSITIONS".UNIT_01.FIXTURE_1.IN_SPARE_STATION_2) OR (("DB8000_PART_STATUS".HMI.PART_STATUS_PART_TYPE_LIST = 2) AND "DB4000_FIX_TABLE_POSITIONS".UNIT_02.FIXTURE_1.IN_MEASURING_STATION_2));
   "DB7235_VARIABLE_LAYOUT".QUALITY.Text[35] := "M_ONE" AND ((("DB8000_PART_STATUS".HMI.PART_STATUS_PART_TYPE_LIST = 1) AND "DB4000_FIX_TABLE_POSITIONS".UNIT_01.FIXTURE_1.IN_SPARE_STATION_2) OR (("DB8000_PART_STATUS".HMI.PART_STATUS_PART_TYPE_LIST = 2) AND "DB4000_FIX_TABLE_POSITIONS".UNIT_02.FIXTURE_1.IN_MEASURING_STATION_2));
   "DB7235_VARIABLE_LAYOUT".QUALITY.Image[2] := "M_ONE" AND ((("DB8000_PART_STATUS".HMI.PART_STATUS_PART_TYPE_LIST = 1) AND "DB4000_FIX_TABLE_POSITIONS".UNIT_01.FIXTURE_1.IN_CLADDING_STATION_3) OR (("DB8000_PART_STATUS".HMI.PART_STATUS_PART_TYPE_LIST = 2) AND "DB4000_FIX_TABLE_POSITIONS".UNIT_02.FIXTURE_1.IN_CLADDING_STATION_3));
   "DB7235_VARIABLE_LAYOUT".QUALITY.Text[36] := "M_ONE" AND ((("DB8000_PART_STATUS".HMI.PART_STATUS_PART_TYPE_LIST = 1) AND "DB4000_FIX_TABLE_POSITIONS".UNIT_01.FIXTURE_1.IN_CLADDING_STATION_3) OR (("DB8000_PART_STATUS".HMI.PART_STATUS_PART_TYPE_LIST = 2) AND "DB4000_FIX_TABLE_POSITIONS".UNIT_02.FIXTURE_1.IN_CLADDING_STATION_3));
   "DB7235_VARIABLE_LAYOUT".QUALITY.Text[31] := "M_ONE" AND ((("DB8000_PART_STATUS".HMI.PART_STATUS_PART_TYPE_LIST = 1) AND "DB4000_FIX_TABLE_POSITIONS".UNIT_01.FIXTURE_1.IN_CLADDING_STATION_3) OR (("DB8000_PART_STATUS".HMI.PART_STATUS_PART_TYPE_LIST = 2) AND "DB4000_FIX_TABLE_POSITIONS".UNIT_02.FIXTURE_1.IN_CLADDING_STATION_3));
   "DB7235_VARIABLE_LAYOUT".QUALITY.Text[29] := "M_ONE" AND ((("DB8000_PART_STATUS".HMI.PART_STATUS_PART_TYPE_LIST = 1) AND "DB4000_FIX_TABLE_POSITIONS".UNIT_01.FIXTURE_1.IN_CLADDING_STATION_3) OR (("DB8000_PART_STATUS".HMI.PART_STATUS_PART_TYPE_LIST = 2) AND "DB4000_FIX_TABLE_POSITIONS".UNIT_02.FIXTURE_1.IN_CLADDING_STATION_3));
   "DB7235_VARIABLE_LAYOUT".QUALITY.Text[39] := "M_ONE" AND ((("DB8000_PART_STATUS".HMI.PART_STATUS_PART_TYPE_LIST = 1) AND "DB4000_FIX_TABLE_POSITIONS".UNIT_01.FIXTURE_1.IN_CLADDING_STATION_3) OR (("DB8000_PART_STATUS".HMI.PART_STATUS_PART_TYPE_LIST = 2) AND "DB4000_FIX_TABLE_POSITIONS".UNIT_02.FIXTURE_1.IN_CLADDING_STATION_3));
   "DB7235_VARIABLE_LAYOUT".QUALITY.Image[3] := "M_ONE" AND ((("DB8000_PART_STATUS".HMI.PART_STATUS_PART_TYPE_LIST = 1) AND "DB4000_FIX_TABLE_POSITIONS".UNIT_01.FIXTURE_1.IN_CLEAN_STATION_4) OR (("DB8000_PART_STATUS".HMI.PART_STATUS_PART_TYPE_LIST = 2) AND "DB4000_FIX_TABLE_POSITIONS".UNIT_02.FIXTURE_1.IN_CLEAN_STATION_4));
   "DB7235_VARIABLE_LAYOUT".QUALITY.Text[38] := "M_ONE" AND ((("DB8000_PART_STATUS".HMI.PART_STATUS_PART_TYPE_LIST = 1) AND "DB4000_FIX_TABLE_POSITIONS".UNIT_01.FIXTURE_1.IN_CLEAN_STATION_4) OR (("DB8000_PART_STATUS".HMI.PART_STATUS_PART_TYPE_LIST = 2) AND "DB4000_FIX_TABLE_POSITIONS".UNIT_02.FIXTURE_1.IN_CLEAN_STATION_4));
   "DB7235_VARIABLE_LAYOUT".QUALITY.Text[34] := "M_ONE" AND ((("DB8000_PART_STATUS".HMI.PART_STATUS_PART_TYPE_LIST = 1) AND "DB4000_FIX_TABLE_POSITIONS".UNIT_01.FIXTURE_1.IN_CLEAN_STATION_4) OR (("DB8000_PART_STATUS".HMI.PART_STATUS_PART_TYPE_LIST = 2) AND "DB4000_FIX_TABLE_POSITIONS".UNIT_02.FIXTURE_1.IN_CLEAN_STATION_4));
   "DB7235_VARIABLE_LAYOUT".QUALITY.Text[27] := "M_ONE" AND ((("DB8000_PART_STATUS".HMI.PART_STATUS_PART_TYPE_LIST = 1) AND "DB4000_FIX_TABLE_POSITIONS".UNIT_01.FIXTURE_1.IN_CLEAN_STATION_4) OR (("DB8000_PART_STATUS".HMI.PART_STATUS_PART_TYPE_LIST = 2) AND "DB4000_FIX_TABLE_POSITIONS".UNIT_02.FIXTURE_1.IN_CLEAN_STATION_4));
   "DB7235_VARIABLE_LAYOUT".QUALITY.Text[30] := "M_ONE" AND ((("DB8000_PART_STATUS".HMI.PART_STATUS_PART_TYPE_LIST = 1) AND "DB4000_FIX_TABLE_POSITIONS".UNIT_01.FIXTURE_1.IN_CLEAN_STATION_4) OR (("DB8000_PART_STATUS".HMI.PART_STATUS_PART_TYPE_LIST = 2) AND "DB4000_FIX_TABLE_POSITIONS".UNIT_02.FIXTURE_1.IN_CLEAN_STATION_4));
   "DB7235_VARIABLE_LAYOUT".QUALITY.Image[4] := "M_ONE" AND ((("DB8000_PART_STATUS".HMI.PART_STATUS_PART_TYPE_LIST = 1) AND "DB4000_FIX_TABLE_POSITIONS".UNIT_01.AXIS_E10_NOT_DEFINED_POS AND NOT "LBP_Axis1".E_NactNmin) OR (("DB8000_PART_STATUS".HMI.PART_STATUS_PART_TYPE_LIST = 2) AND "DB4000_FIX_TABLE_POSITIONS".UNIT_02.AXIS_E20_NOT_DEFINED_POS AND NOT "LBP_Axis15".E_NactNmin));
END_REGION

REGION Network 13: PART STATUS UNIT 02
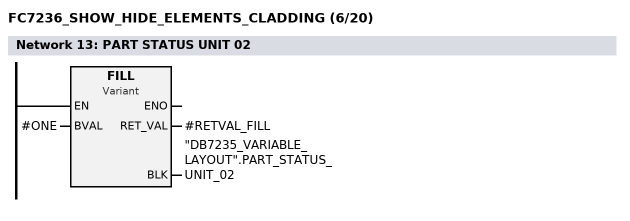
   RUNG wire#powerrail
      { S7_Templates := "ptr_type := Variant" } FILL(BVAL := #ONE, RET_VAL => #RETVAL_FILL, BLK => "DB7235_VARIABLE_LAYOUT".PART_STATUS_UNIT_02)
   END_RUNG
   // the same network as SCL:
   #RETVAL_FILL := FILL(BVAL := #ONE, BLK => "DB7235_VARIABLE_LAYOUT".PART_STATUS_UNIT_02);
END_REGION

REGION Network 14: PART STATUS IO FIELD AND TEXTS UNIT 02
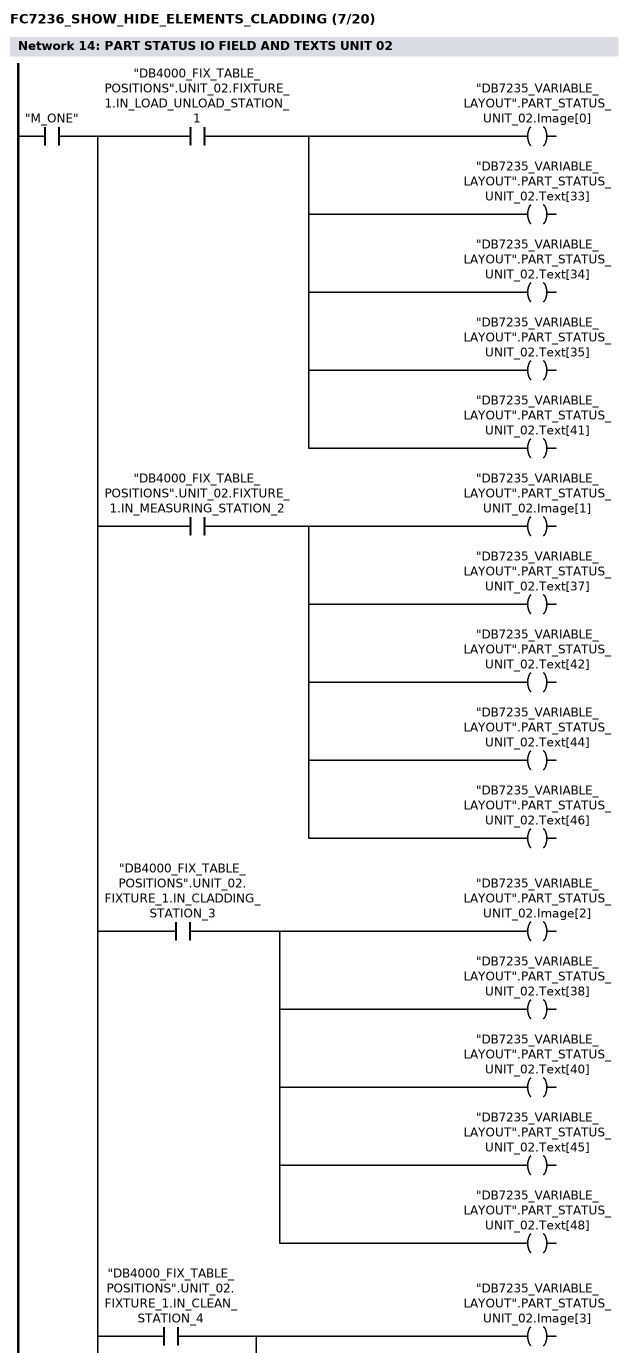
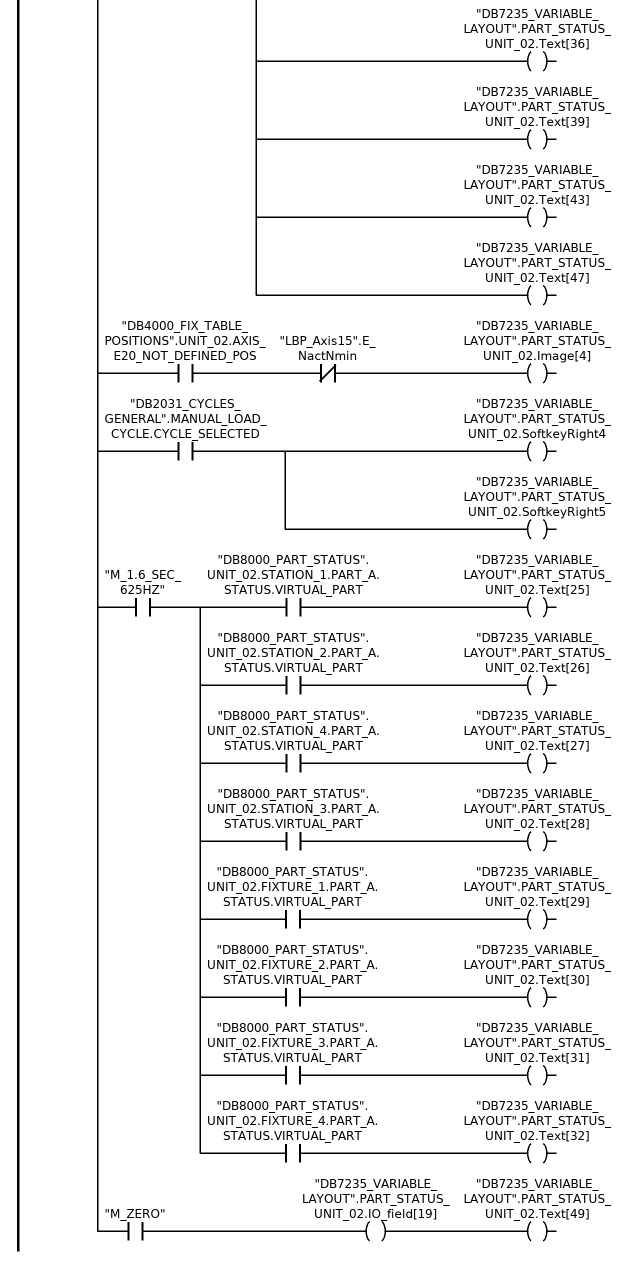
   RUNG wire#powerrail
      Contact( "M_ONE" )
      wire#w1
      Contact( "DB4000_FIX_TABLE_POSITIONS".UNIT_02.FIXTURE_1.IN_LOAD_UNLOAD_STATION_1 )
      wire#w2
      Coil( "DB7235_VARIABLE_LAYOUT".PART_STATUS_UNIT_02.Image[0] )
   END_RUNG
   RUNG wire#w2
      Coil( "DB7235_VARIABLE_LAYOUT".PART_STATUS_UNIT_02.Text[33] )
   END_RUNG
   RUNG wire#w2
      Coil( "DB7235_VARIABLE_LAYOUT".PART_STATUS_UNIT_02.Text[34] )
   END_RUNG
   RUNG wire#w2
      Coil( "DB7235_VARIABLE_LAYOUT".PART_STATUS_UNIT_02.Text[35] )
   END_RUNG
   RUNG wire#w2
      Coil( "DB7235_VARIABLE_LAYOUT".PART_STATUS_UNIT_02.Text[41] )
   END_RUNG
   RUNG wire#w1
      Contact( "DB4000_FIX_TABLE_POSITIONS".UNIT_02.FIXTURE_1.IN_MEASURING_STATION_2 )
      wire#w3
      Coil( "DB7235_VARIABLE_LAYOUT".PART_STATUS_UNIT_02.Image[1] )
   END_RUNG
   RUNG wire#w3
      Coil( "DB7235_VARIABLE_LAYOUT".PART_STATUS_UNIT_02.Text[37] )
   END_RUNG
   RUNG wire#w3
      Coil( "DB7235_VARIABLE_LAYOUT".PART_STATUS_UNIT_02.Text[42] )
   END_RUNG
   RUNG wire#w3
      Coil( "DB7235_VARIABLE_LAYOUT".PART_STATUS_UNIT_02.Text[44] )
   END_RUNG
   RUNG wire#w3
      Coil( "DB7235_VARIABLE_LAYOUT".PART_STATUS_UNIT_02.Text[46] )
   END_RUNG
   RUNG wire#w1
      Contact( "DB4000_FIX_TABLE_POSITIONS".UNIT_02.FIXTURE_1.IN_CLADDING_STATION_3 )
      wire#w4
      Coil( "DB7235_VARIABLE_LAYOUT".PART_STATUS_UNIT_02.Image[2] )
   END_RUNG
   RUNG wire#w4
      Coil( "DB7235_VARIABLE_LAYOUT".PART_STATUS_UNIT_02.Text[38] )
   END_RUNG
   RUNG wire#w4
      Coil( "DB7235_VARIABLE_LAYOUT".PART_STATUS_UNIT_02.Text[40] )
   END_RUNG
   RUNG wire#w4
      Coil( "DB7235_VARIABLE_LAYOUT".PART_STATUS_UNIT_02.Text[45] )
   END_RUNG
   RUNG wire#w4
      Coil( "DB7235_VARIABLE_LAYOUT".PART_STATUS_UNIT_02.Text[48] )
   END_RUNG
   RUNG wire#w1
      Contact( "DB4000_FIX_TABLE_POSITIONS".UNIT_02.FIXTURE_1.IN_CLEAN_STATION_4 )
      wire#w5
      Coil( "DB7235_VARIABLE_LAYOUT".PART_STATUS_UNIT_02.Image[3] )
   END_RUNG
   RUNG wire#w5
      Coil( "DB7235_VARIABLE_LAYOUT".PART_STATUS_UNIT_02.Text[36] )
   END_RUNG
   RUNG wire#w5
      Coil( "DB7235_VARIABLE_LAYOUT".PART_STATUS_UNIT_02.Text[39] )
   END_RUNG
   RUNG wire#w5
      Coil( "DB7235_VARIABLE_LAYOUT".PART_STATUS_UNIT_02.Text[43] )
   END_RUNG
   RUNG wire#w5
      Coil( "DB7235_VARIABLE_LAYOUT".PART_STATUS_UNIT_02.Text[47] )
   END_RUNG
   RUNG wire#w1
      Contact( "DB4000_FIX_TABLE_POSITIONS".UNIT_02.AXIS_E20_NOT_DEFINED_POS )
      I_Contact( "LBP_Axis15".E_NactNmin )
      Coil( "DB7235_VARIABLE_LAYOUT".PART_STATUS_UNIT_02.Image[4] )
   END_RUNG
   RUNG wire#w1
      Contact( "DB2031_CYCLES_GENERAL".MANUAL_LOAD_CYCLE.CYCLE_SELECTED )
      wire#w6
      Coil( "DB7235_VARIABLE_LAYOUT".PART_STATUS_UNIT_02.SoftkeyRight4 )
   END_RUNG
   RUNG wire#w6
      Coil( "DB7235_VARIABLE_LAYOUT".PART_STATUS_UNIT_02.SoftkeyRight5 )
   END_RUNG
   RUNG wire#w1
      Contact( "M_1.6_SEC_625HZ" )
      wire#w7
      Contact( "DB8000_PART_STATUS".UNIT_02.STATION_1.PART_A.STATUS.VIRTUAL_PART )
      Coil( "DB7235_VARIABLE_LAYOUT".PART_STATUS_UNIT_02.Text[25] )
   END_RUNG
   RUNG wire#w7
      Contact( "DB8000_PART_STATUS".UNIT_02.STATION_2.PART_A.STATUS.VIRTUAL_PART )
      Coil( "DB7235_VARIABLE_LAYOUT".PART_STATUS_UNIT_02.Text[26] )
   END_RUNG
   RUNG wire#w7
      Contact( "DB8000_PART_STATUS".UNIT_02.STATION_4.PART_A.STATUS.VIRTUAL_PART )
      Coil( "DB7235_VARIABLE_LAYOUT".PART_STATUS_UNIT_02.Text[27] )
   END_RUNG
   RUNG wire#w7
      Contact( "DB8000_PART_STATUS".UNIT_02.STATION_3.PART_A.STATUS.VIRTUAL_PART )
      Coil( "DB7235_VARIABLE_LAYOUT".PART_STATUS_UNIT_02.Text[28] )
   END_RUNG
   RUNG wire#w7
      Contact( "DB8000_PART_STATUS".UNIT_02.FIXTURE_1.PART_A.STATUS.VIRTUAL_PART )
      Coil( "DB7235_VARIABLE_LAYOUT".PART_STATUS_UNIT_02.Text[29] )
   END_RUNG
   RUNG wire#w7
      Contact( "DB8000_PART_STATUS".UNIT_02.FIXTURE_2.PART_A.STATUS.VIRTUAL_PART )
      Coil( "DB7235_VARIABLE_LAYOUT".PART_STATUS_UNIT_02.Text[30] )
   END_RUNG
   RUNG wire#w7
      Contact( "DB8000_PART_STATUS".UNIT_02.FIXTURE_3.PART_A.STATUS.VIRTUAL_PART )
      Coil( "DB7235_VARIABLE_LAYOUT".PART_STATUS_UNIT_02.Text[31] )
   END_RUNG
   RUNG wire#w7
      Contact( "DB8000_PART_STATUS".UNIT_02.FIXTURE_4.PART_A.STATUS.VIRTUAL_PART )
      Coil( "DB7235_VARIABLE_LAYOUT".PART_STATUS_UNIT_02.Text[32] )
   END_RUNG
   RUNG wire#w1
      Contact( "M_ZERO" )
      Coil( "DB7235_VARIABLE_LAYOUT".PART_STATUS_UNIT_02.IO_field[19] )
      Coil( "DB7235_VARIABLE_LAYOUT".PART_STATUS_UNIT_02.Text[49] )
   END_RUNG
   // the same network as SCL:
   "DB7235_VARIABLE_LAYOUT".PART_STATUS_UNIT_02.Image[0] := "M_ONE" AND "DB4000_FIX_TABLE_POSITIONS".UNIT_02.FIXTURE_1.IN_LOAD_UNLOAD_STATION_1;
   "DB7235_VARIABLE_LAYOUT".PART_STATUS_UNIT_02.Text[33] := "M_ONE" AND "DB4000_FIX_TABLE_POSITIONS".UNIT_02.FIXTURE_1.IN_LOAD_UNLOAD_STATION_1;
   "DB7235_VARIABLE_LAYOUT".PART_STATUS_UNIT_02.Text[34] := "M_ONE" AND "DB4000_FIX_TABLE_POSITIONS".UNIT_02.FIXTURE_1.IN_LOAD_UNLOAD_STATION_1;
   "DB7235_VARIABLE_LAYOUT".PART_STATUS_UNIT_02.Text[35] := "M_ONE" AND "DB4000_FIX_TABLE_POSITIONS".UNIT_02.FIXTURE_1.IN_LOAD_UNLOAD_STATION_1;
   "DB7235_VARIABLE_LAYOUT".PART_STATUS_UNIT_02.Text[41] := "M_ONE" AND "DB4000_FIX_TABLE_POSITIONS".UNIT_02.FIXTURE_1.IN_LOAD_UNLOAD_STATION_1;
   "DB7235_VARIABLE_LAYOUT".PART_STATUS_UNIT_02.Image[1] := "M_ONE" AND "DB4000_FIX_TABLE_POSITIONS".UNIT_02.FIXTURE_1.IN_MEASURING_STATION_2;
   "DB7235_VARIABLE_LAYOUT".PART_STATUS_UNIT_02.Text[37] := "M_ONE" AND "DB4000_FIX_TABLE_POSITIONS".UNIT_02.FIXTURE_1.IN_MEASURING_STATION_2;
   "DB7235_VARIABLE_LAYOUT".PART_STATUS_UNIT_02.Text[42] := "M_ONE" AND "DB4000_FIX_TABLE_POSITIONS".UNIT_02.FIXTURE_1.IN_MEASURING_STATION_2;
   "DB7235_VARIABLE_LAYOUT".PART_STATUS_UNIT_02.Text[44] := "M_ONE" AND "DB4000_FIX_TABLE_POSITIONS".UNIT_02.FIXTURE_1.IN_MEASURING_STATION_2;
   "DB7235_VARIABLE_LAYOUT".PART_STATUS_UNIT_02.Text[46] := "M_ONE" AND "DB4000_FIX_TABLE_POSITIONS".UNIT_02.FIXTURE_1.IN_MEASURING_STATION_2;
   "DB7235_VARIABLE_LAYOUT".PART_STATUS_UNIT_02.Image[2] := "M_ONE" AND "DB4000_FIX_TABLE_POSITIONS".UNIT_02.FIXTURE_1.IN_CLADDING_STATION_3;
   "DB7235_VARIABLE_LAYOUT".PART_STATUS_UNIT_02.Text[38] := "M_ONE" AND "DB4000_FIX_TABLE_POSITIONS".UNIT_02.FIXTURE_1.IN_CLADDING_STATION_3;
   "DB7235_VARIABLE_LAYOUT".PART_STATUS_UNIT_02.Text[40] := "M_ONE" AND "DB4000_FIX_TABLE_POSITIONS".UNIT_02.FIXTURE_1.IN_CLADDING_STATION_3;
   "DB7235_VARIABLE_LAYOUT".PART_STATUS_UNIT_02.Text[45] := "M_ONE" AND "DB4000_FIX_TABLE_POSITIONS".UNIT_02.FIXTURE_1.IN_CLADDING_STATION_3;
   "DB7235_VARIABLE_LAYOUT".PART_STATUS_UNIT_02.Text[48] := "M_ONE" AND "DB4000_FIX_TABLE_POSITIONS".UNIT_02.FIXTURE_1.IN_CLADDING_STATION_3;
   "DB7235_VARIABLE_LAYOUT".PART_STATUS_UNIT_02.Image[3] := "M_ONE" AND "DB4000_FIX_TABLE_POSITIONS".UNIT_02.FIXTURE_1.IN_CLEAN_STATION_4;
   "DB7235_VARIABLE_LAYOUT".PART_STATUS_UNIT_02.Text[36] := "M_ONE" AND "DB4000_FIX_TABLE_POSITIONS".UNIT_02.FIXTURE_1.IN_CLEAN_STATION_4;
   "DB7235_VARIABLE_LAYOUT".PART_STATUS_UNIT_02.Text[39] := "M_ONE" AND "DB4000_FIX_TABLE_POSITIONS".UNIT_02.FIXTURE_1.IN_CLEAN_STATION_4;
   "DB7235_VARIABLE_LAYOUT".PART_STATUS_UNIT_02.Text[43] := "M_ONE" AND "DB4000_FIX_TABLE_POSITIONS".UNIT_02.FIXTURE_1.IN_CLEAN_STATION_4;
   "DB7235_VARIABLE_LAYOUT".PART_STATUS_UNIT_02.Text[47] := "M_ONE" AND "DB4000_FIX_TABLE_POSITIONS".UNIT_02.FIXTURE_1.IN_CLEAN_STATION_4;
   "DB7235_VARIABLE_LAYOUT".PART_STATUS_UNIT_02.Image[4] := "M_ONE" AND "DB4000_FIX_TABLE_POSITIONS".UNIT_02.AXIS_E20_NOT_DEFINED_POS AND NOT "LBP_Axis15".E_NactNmin;
   "DB7235_VARIABLE_LAYOUT".PART_STATUS_UNIT_02.SoftkeyRight4 := "M_ONE" AND "DB2031_CYCLES_GENERAL".MANUAL_LOAD_CYCLE.CYCLE_SELECTED;
   "DB7235_VARIABLE_LAYOUT".PART_STATUS_UNIT_02.SoftkeyRight5 := "DB7235_VARIABLE_LAYOUT".PART_STATUS_UNIT_02.SoftkeyRight4;
   #_w1 := "M_ONE" AND "M_1.6_SEC_625HZ";
   "DB7235_VARIABLE_LAYOUT".PART_STATUS_UNIT_02.Text[25] := #_w1 AND "DB8000_PART_STATUS".UNIT_02.STATION_1.PART_A.STATUS.VIRTUAL_PART;
   "DB7235_VARIABLE_LAYOUT".PART_STATUS_UNIT_02.Text[26] := #_w1 AND "DB8000_PART_STATUS".UNIT_02.STATION_2.PART_A.STATUS.VIRTUAL_PART;
   "DB7235_VARIABLE_LAYOUT".PART_STATUS_UNIT_02.Text[27] := #_w1 AND "DB8000_PART_STATUS".UNIT_02.STATION_4.PART_A.STATUS.VIRTUAL_PART;
   "DB7235_VARIABLE_LAYOUT".PART_STATUS_UNIT_02.Text[28] := #_w1 AND "DB8000_PART_STATUS".UNIT_02.STATION_3.PART_A.STATUS.VIRTUAL_PART;
   "DB7235_VARIABLE_LAYOUT".PART_STATUS_UNIT_02.Text[29] := #_w1 AND "DB8000_PART_STATUS".UNIT_02.FIXTURE_1.PART_A.STATUS.VIRTUAL_PART;
   "DB7235_VARIABLE_LAYOUT".PART_STATUS_UNIT_02.Text[30] := #_w1 AND "DB8000_PART_STATUS".UNIT_02.FIXTURE_2.PART_A.STATUS.VIRTUAL_PART;
   "DB7235_VARIABLE_LAYOUT".PART_STATUS_UNIT_02.Text[31] := #_w1 AND "DB8000_PART_STATUS".UNIT_02.FIXTURE_3.PART_A.STATUS.VIRTUAL_PART;
   "DB7235_VARIABLE_LAYOUT".PART_STATUS_UNIT_02.Text[32] := #_w1 AND "DB8000_PART_STATUS".UNIT_02.FIXTURE_4.PART_A.STATUS.VIRTUAL_PART;
   "DB7235_VARIABLE_LAYOUT".PART_STATUS_UNIT_02.IO_field[19] := "M_ONE" AND "M_ZERO";
   "DB7235_VARIABLE_LAYOUT".PART_STATUS_UNIT_02.Text[49] := "M_ONE" AND "M_ZERO";
END_REGION

REGION Network 15: PART ID UNIT 01
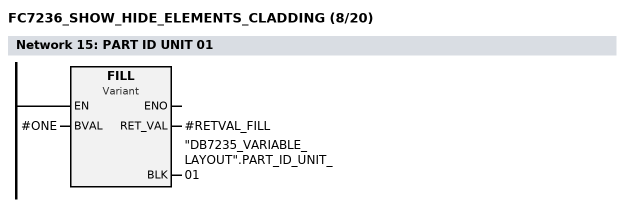
   RUNG wire#powerrail
      { S7_Templates := "ptr_type := Variant" } FILL(BVAL := #ONE, RET_VAL => #RETVAL_FILL, BLK => "DB7235_VARIABLE_LAYOUT".PART_ID_UNIT_01)
   END_RUNG
   // the same network as SCL:
   #RETVAL_FILL := FILL(BVAL := #ONE, BLK => "DB7235_VARIABLE_LAYOUT".PART_ID_UNIT_01);
END_REGION

REGION Network 16: PART ID IO FIELD AND TEXTS UNIT 01
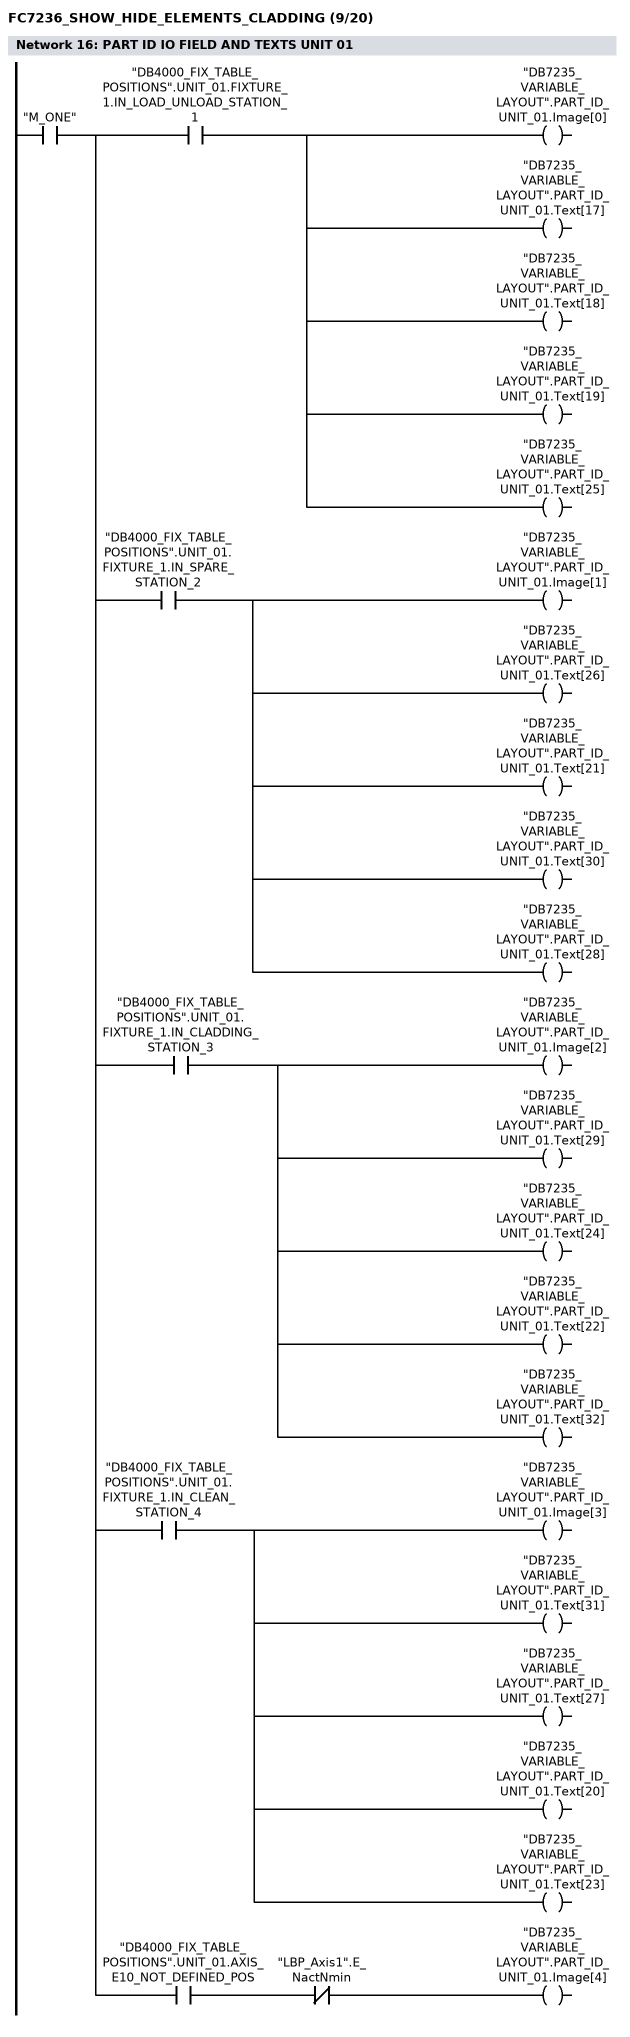
   RUNG wire#powerrail
      Contact( "M_ONE" )
      wire#w1
      Contact( "DB4000_FIX_TABLE_POSITIONS".UNIT_01.FIXTURE_1.IN_LOAD_UNLOAD_STATION_1 )
      wire#w2
      Coil( "DB7235_VARIABLE_LAYOUT".PART_ID_UNIT_01.Image[0] )
   END_RUNG
   RUNG wire#w2
      Coil( "DB7235_VARIABLE_LAYOUT".PART_ID_UNIT_01.Text[17] )
   END_RUNG
   RUNG wire#w2
      Coil( "DB7235_VARIABLE_LAYOUT".PART_ID_UNIT_01.Text[18] )
   END_RUNG
   RUNG wire#w2
      Coil( "DB7235_VARIABLE_LAYOUT".PART_ID_UNIT_01.Text[19] )
   END_RUNG
   RUNG wire#w2
      Coil( "DB7235_VARIABLE_LAYOUT".PART_ID_UNIT_01.Text[25] )
   END_RUNG
   RUNG wire#w1
      Contact( "DB4000_FIX_TABLE_POSITIONS".UNIT_01.FIXTURE_1.IN_SPARE_STATION_2 )
      wire#w3
      Coil( "DB7235_VARIABLE_LAYOUT".PART_ID_UNIT_01.Image[1] )
   END_RUNG
   RUNG wire#w3
      Coil( "DB7235_VARIABLE_LAYOUT".PART_ID_UNIT_01.Text[26] )
   END_RUNG
   RUNG wire#w3
      Coil( "DB7235_VARIABLE_LAYOUT".PART_ID_UNIT_01.Text[21] )
   END_RUNG
   RUNG wire#w3
      Coil( "DB7235_VARIABLE_LAYOUT".PART_ID_UNIT_01.Text[30] )
   END_RUNG
   RUNG wire#w3
      Coil( "DB7235_VARIABLE_LAYOUT".PART_ID_UNIT_01.Text[28] )
   END_RUNG
   RUNG wire#w1
      Contact( "DB4000_FIX_TABLE_POSITIONS".UNIT_01.FIXTURE_1.IN_CLADDING_STATION_3 )
      wire#w4
      Coil( "DB7235_VARIABLE_LAYOUT".PART_ID_UNIT_01.Image[2] )
   END_RUNG
   RUNG wire#w4
      Coil( "DB7235_VARIABLE_LAYOUT".PART_ID_UNIT_01.Text[29] )
   END_RUNG
   RUNG wire#w4
      Coil( "DB7235_VARIABLE_LAYOUT".PART_ID_UNIT_01.Text[24] )
   END_RUNG
   RUNG wire#w4
      Coil( "DB7235_VARIABLE_LAYOUT".PART_ID_UNIT_01.Text[22] )
   END_RUNG
   RUNG wire#w4
      Coil( "DB7235_VARIABLE_LAYOUT".PART_ID_UNIT_01.Text[32] )
   END_RUNG
   RUNG wire#w1
      Contact( "DB4000_FIX_TABLE_POSITIONS".UNIT_01.FIXTURE_1.IN_CLEAN_STATION_4 )
      wire#w5
      Coil( "DB7235_VARIABLE_LAYOUT".PART_ID_UNIT_01.Image[3] )
   END_RUNG
   RUNG wire#w5
      Coil( "DB7235_VARIABLE_LAYOUT".PART_ID_UNIT_01.Text[31] )
   END_RUNG
   RUNG wire#w5
      Coil( "DB7235_VARIABLE_LAYOUT".PART_ID_UNIT_01.Text[27] )
   END_RUNG
   RUNG wire#w5
      Coil( "DB7235_VARIABLE_LAYOUT".PART_ID_UNIT_01.Text[20] )
   END_RUNG
   RUNG wire#w5
      Coil( "DB7235_VARIABLE_LAYOUT".PART_ID_UNIT_01.Text[23] )
   END_RUNG
   RUNG wire#w1
      Contact( "DB4000_FIX_TABLE_POSITIONS".UNIT_01.AXIS_E10_NOT_DEFINED_POS )
      I_Contact( "LBP_Axis1".E_NactNmin )
      Coil( "DB7235_VARIABLE_LAYOUT".PART_ID_UNIT_01.Image[4] )
   END_RUNG
   // the same network as SCL:
   "DB7235_VARIABLE_LAYOUT".PART_ID_UNIT_01.Image[0] := "M_ONE" AND "DB4000_FIX_TABLE_POSITIONS".UNIT_01.FIXTURE_1.IN_LOAD_UNLOAD_STATION_1;
   "DB7235_VARIABLE_LAYOUT".PART_ID_UNIT_01.Text[17] := "M_ONE" AND "DB4000_FIX_TABLE_POSITIONS".UNIT_01.FIXTURE_1.IN_LOAD_UNLOAD_STATION_1;
   "DB7235_VARIABLE_LAYOUT".PART_ID_UNIT_01.Text[18] := "M_ONE" AND "DB4000_FIX_TABLE_POSITIONS".UNIT_01.FIXTURE_1.IN_LOAD_UNLOAD_STATION_1;
   "DB7235_VARIABLE_LAYOUT".PART_ID_UNIT_01.Text[19] := "M_ONE" AND "DB4000_FIX_TABLE_POSITIONS".UNIT_01.FIXTURE_1.IN_LOAD_UNLOAD_STATION_1;
   "DB7235_VARIABLE_LAYOUT".PART_ID_UNIT_01.Text[25] := "M_ONE" AND "DB4000_FIX_TABLE_POSITIONS".UNIT_01.FIXTURE_1.IN_LOAD_UNLOAD_STATION_1;
   "DB7235_VARIABLE_LAYOUT".PART_ID_UNIT_01.Image[1] := "M_ONE" AND "DB4000_FIX_TABLE_POSITIONS".UNIT_01.FIXTURE_1.IN_SPARE_STATION_2;
   "DB7235_VARIABLE_LAYOUT".PART_ID_UNIT_01.Text[26] := "M_ONE" AND "DB4000_FIX_TABLE_POSITIONS".UNIT_01.FIXTURE_1.IN_SPARE_STATION_2;
   "DB7235_VARIABLE_LAYOUT".PART_ID_UNIT_01.Text[21] := "M_ONE" AND "DB4000_FIX_TABLE_POSITIONS".UNIT_01.FIXTURE_1.IN_SPARE_STATION_2;
   "DB7235_VARIABLE_LAYOUT".PART_ID_UNIT_01.Text[30] := "M_ONE" AND "DB4000_FIX_TABLE_POSITIONS".UNIT_01.FIXTURE_1.IN_SPARE_STATION_2;
   "DB7235_VARIABLE_LAYOUT".PART_ID_UNIT_01.Text[28] := "M_ONE" AND "DB4000_FIX_TABLE_POSITIONS".UNIT_01.FIXTURE_1.IN_SPARE_STATION_2;
   "DB7235_VARIABLE_LAYOUT".PART_ID_UNIT_01.Image[2] := "M_ONE" AND "DB4000_FIX_TABLE_POSITIONS".UNIT_01.FIXTURE_1.IN_CLADDING_STATION_3;
   "DB7235_VARIABLE_LAYOUT".PART_ID_UNIT_01.Text[29] := "M_ONE" AND "DB4000_FIX_TABLE_POSITIONS".UNIT_01.FIXTURE_1.IN_CLADDING_STATION_3;
   "DB7235_VARIABLE_LAYOUT".PART_ID_UNIT_01.Text[24] := "M_ONE" AND "DB4000_FIX_TABLE_POSITIONS".UNIT_01.FIXTURE_1.IN_CLADDING_STATION_3;
   "DB7235_VARIABLE_LAYOUT".PART_ID_UNIT_01.Text[22] := "M_ONE" AND "DB4000_FIX_TABLE_POSITIONS".UNIT_01.FIXTURE_1.IN_CLADDING_STATION_3;
   "DB7235_VARIABLE_LAYOUT".PART_ID_UNIT_01.Text[32] := "M_ONE" AND "DB4000_FIX_TABLE_POSITIONS".UNIT_01.FIXTURE_1.IN_CLADDING_STATION_3;
   "DB7235_VARIABLE_LAYOUT".PART_ID_UNIT_01.Image[3] := "M_ONE" AND "DB4000_FIX_TABLE_POSITIONS".UNIT_01.FIXTURE_1.IN_CLEAN_STATION_4;
   "DB7235_VARIABLE_LAYOUT".PART_ID_UNIT_01.Text[31] := "M_ONE" AND "DB4000_FIX_TABLE_POSITIONS".UNIT_01.FIXTURE_1.IN_CLEAN_STATION_4;
   "DB7235_VARIABLE_LAYOUT".PART_ID_UNIT_01.Text[27] := "M_ONE" AND "DB4000_FIX_TABLE_POSITIONS".UNIT_01.FIXTURE_1.IN_CLEAN_STATION_4;
   "DB7235_VARIABLE_LAYOUT".PART_ID_UNIT_01.Text[20] := "M_ONE" AND "DB4000_FIX_TABLE_POSITIONS".UNIT_01.FIXTURE_1.IN_CLEAN_STATION_4;
   "DB7235_VARIABLE_LAYOUT".PART_ID_UNIT_01.Text[23] := "M_ONE" AND "DB4000_FIX_TABLE_POSITIONS".UNIT_01.FIXTURE_1.IN_CLEAN_STATION_4;
   "DB7235_VARIABLE_LAYOUT".PART_ID_UNIT_01.Image[4] := "M_ONE" AND "DB4000_FIX_TABLE_POSITIONS".UNIT_01.AXIS_E10_NOT_DEFINED_POS AND NOT "LBP_Axis1".E_NactNmin;
END_REGION

REGION Network 17: PART ID UNIT 02
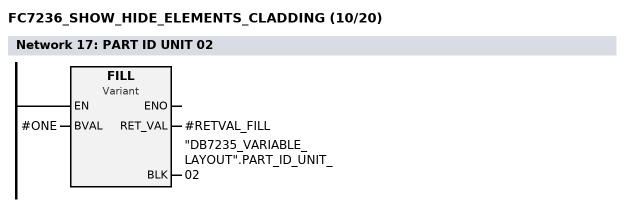
   RUNG wire#powerrail
      { S7_Templates := "ptr_type := Variant" } FILL(BVAL := #ONE, RET_VAL => #RETVAL_FILL, BLK => "DB7235_VARIABLE_LAYOUT".PART_ID_UNIT_02)
   END_RUNG
   // the same network as SCL:
   #RETVAL_FILL := FILL(BVAL := #ONE, BLK => "DB7235_VARIABLE_LAYOUT".PART_ID_UNIT_02);
END_REGION

REGION Network 18: PART ID IO FIELD AND TEXTS UNIT 02
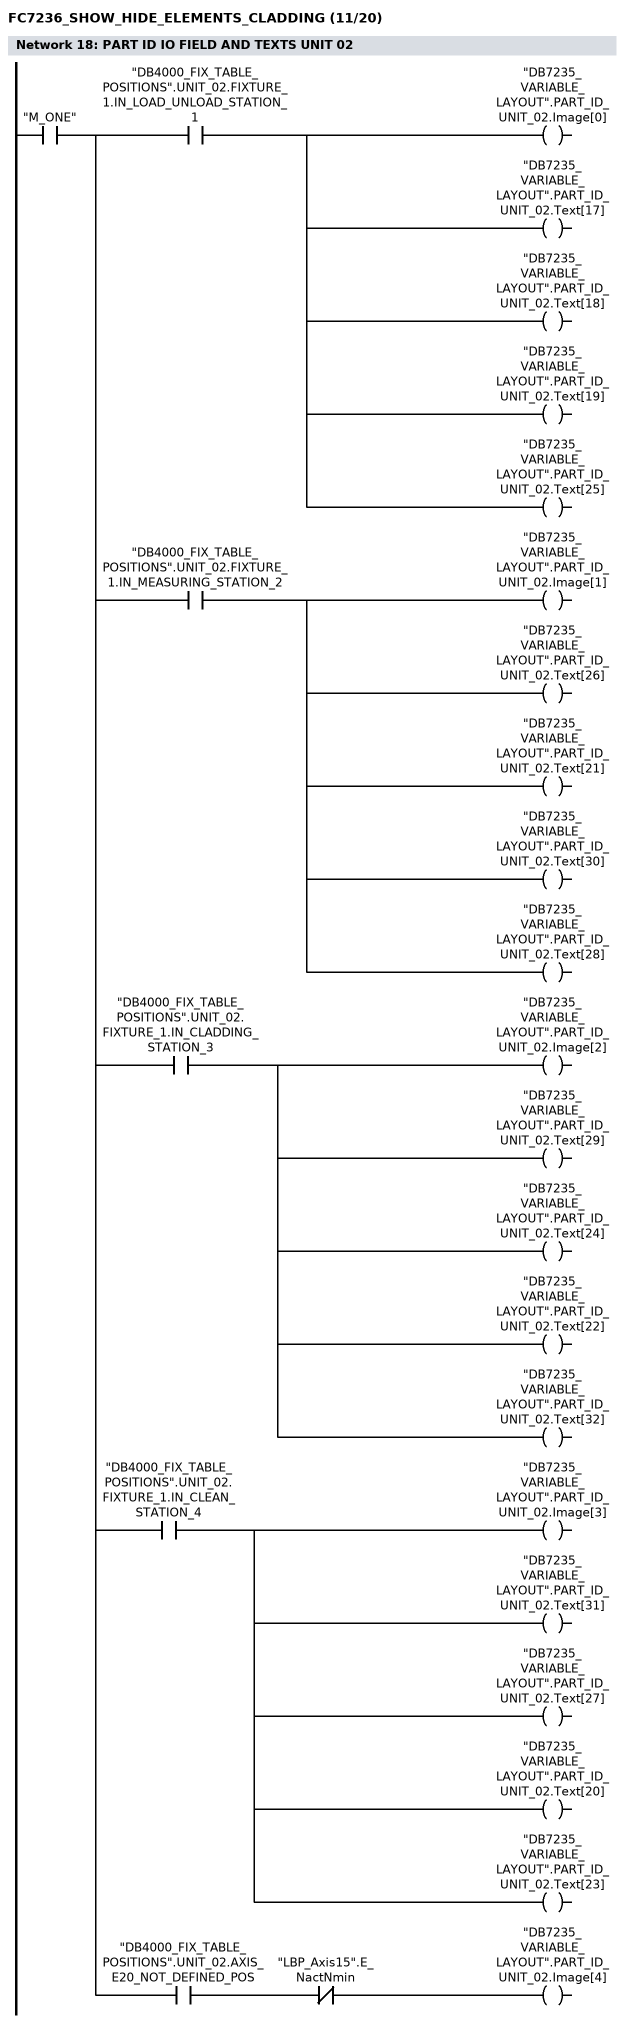
   RUNG wire#powerrail
      Contact( "M_ONE" )
      wire#w1
      Contact( "DB4000_FIX_TABLE_POSITIONS".UNIT_02.FIXTURE_1.IN_LOAD_UNLOAD_STATION_1 )
      wire#w2
      Coil( "DB7235_VARIABLE_LAYOUT".PART_ID_UNIT_02.Image[0] )
   END_RUNG
   RUNG wire#w2
      Coil( "DB7235_VARIABLE_LAYOUT".PART_ID_UNIT_02.Text[17] )
   END_RUNG
   RUNG wire#w2
      Coil( "DB7235_VARIABLE_LAYOUT".PART_ID_UNIT_02.Text[18] )
   END_RUNG
   RUNG wire#w2
      Coil( "DB7235_VARIABLE_LAYOUT".PART_ID_UNIT_02.Text[19] )
   END_RUNG
   RUNG wire#w2
      Coil( "DB7235_VARIABLE_LAYOUT".PART_ID_UNIT_02.Text[25] )
   END_RUNG
   RUNG wire#w1
      Contact( "DB4000_FIX_TABLE_POSITIONS".UNIT_02.FIXTURE_1.IN_MEASURING_STATION_2 )
      wire#w3
      Coil( "DB7235_VARIABLE_LAYOUT".PART_ID_UNIT_02.Image[1] )
   END_RUNG
   RUNG wire#w3
      Coil( "DB7235_VARIABLE_LAYOUT".PART_ID_UNIT_02.Text[26] )
   END_RUNG
   RUNG wire#w3
      Coil( "DB7235_VARIABLE_LAYOUT".PART_ID_UNIT_02.Text[21] )
   END_RUNG
   RUNG wire#w3
      Coil( "DB7235_VARIABLE_LAYOUT".PART_ID_UNIT_02.Text[30] )
   END_RUNG
   RUNG wire#w3
      Coil( "DB7235_VARIABLE_LAYOUT".PART_ID_UNIT_02.Text[28] )
   END_RUNG
   RUNG wire#w1
      Contact( "DB4000_FIX_TABLE_POSITIONS".UNIT_02.FIXTURE_1.IN_CLADDING_STATION_3 )
      wire#w4
      Coil( "DB7235_VARIABLE_LAYOUT".PART_ID_UNIT_02.Image[2] )
   END_RUNG
   RUNG wire#w4
      Coil( "DB7235_VARIABLE_LAYOUT".PART_ID_UNIT_02.Text[29] )
   END_RUNG
   RUNG wire#w4
      Coil( "DB7235_VARIABLE_LAYOUT".PART_ID_UNIT_02.Text[24] )
   END_RUNG
   RUNG wire#w4
      Coil( "DB7235_VARIABLE_LAYOUT".PART_ID_UNIT_02.Text[22] )
   END_RUNG
   RUNG wire#w4
      Coil( "DB7235_VARIABLE_LAYOUT".PART_ID_UNIT_02.Text[32] )
   END_RUNG
   RUNG wire#w1
      Contact( "DB4000_FIX_TABLE_POSITIONS".UNIT_02.FIXTURE_1.IN_CLEAN_STATION_4 )
      wire#w5
      Coil( "DB7235_VARIABLE_LAYOUT".PART_ID_UNIT_02.Image[3] )
   END_RUNG
   RUNG wire#w5
      Coil( "DB7235_VARIABLE_LAYOUT".PART_ID_UNIT_02.Text[31] )
   END_RUNG
   RUNG wire#w5
      Coil( "DB7235_VARIABLE_LAYOUT".PART_ID_UNIT_02.Text[27] )
   END_RUNG
   RUNG wire#w5
      Coil( "DB7235_VARIABLE_LAYOUT".PART_ID_UNIT_02.Text[20] )
   END_RUNG
   RUNG wire#w5
      Coil( "DB7235_VARIABLE_LAYOUT".PART_ID_UNIT_02.Text[23] )
   END_RUNG
   RUNG wire#w1
      Contact( "DB4000_FIX_TABLE_POSITIONS".UNIT_02.AXIS_E20_NOT_DEFINED_POS )
      I_Contact( "LBP_Axis15".E_NactNmin )
      Coil( "DB7235_VARIABLE_LAYOUT".PART_ID_UNIT_02.Image[4] )
   END_RUNG
   // the same network as SCL:
   "DB7235_VARIABLE_LAYOUT".PART_ID_UNIT_02.Image[0] := "M_ONE" AND "DB4000_FIX_TABLE_POSITIONS".UNIT_02.FIXTURE_1.IN_LOAD_UNLOAD_STATION_1;
   "DB7235_VARIABLE_LAYOUT".PART_ID_UNIT_02.Text[17] := "M_ONE" AND "DB4000_FIX_TABLE_POSITIONS".UNIT_02.FIXTURE_1.IN_LOAD_UNLOAD_STATION_1;
   "DB7235_VARIABLE_LAYOUT".PART_ID_UNIT_02.Text[18] := "M_ONE" AND "DB4000_FIX_TABLE_POSITIONS".UNIT_02.FIXTURE_1.IN_LOAD_UNLOAD_STATION_1;
   "DB7235_VARIABLE_LAYOUT".PART_ID_UNIT_02.Text[19] := "M_ONE" AND "DB4000_FIX_TABLE_POSITIONS".UNIT_02.FIXTURE_1.IN_LOAD_UNLOAD_STATION_1;
   "DB7235_VARIABLE_LAYOUT".PART_ID_UNIT_02.Text[25] := "M_ONE" AND "DB4000_FIX_TABLE_POSITIONS".UNIT_02.FIXTURE_1.IN_LOAD_UNLOAD_STATION_1;
   "DB7235_VARIABLE_LAYOUT".PART_ID_UNIT_02.Image[1] := "M_ONE" AND "DB4000_FIX_TABLE_POSITIONS".UNIT_02.FIXTURE_1.IN_MEASURING_STATION_2;
   "DB7235_VARIABLE_LAYOUT".PART_ID_UNIT_02.Text[26] := "M_ONE" AND "DB4000_FIX_TABLE_POSITIONS".UNIT_02.FIXTURE_1.IN_MEASURING_STATION_2;
   "DB7235_VARIABLE_LAYOUT".PART_ID_UNIT_02.Text[21] := "M_ONE" AND "DB4000_FIX_TABLE_POSITIONS".UNIT_02.FIXTURE_1.IN_MEASURING_STATION_2;
   "DB7235_VARIABLE_LAYOUT".PART_ID_UNIT_02.Text[30] := "M_ONE" AND "DB4000_FIX_TABLE_POSITIONS".UNIT_02.FIXTURE_1.IN_MEASURING_STATION_2;
   "DB7235_VARIABLE_LAYOUT".PART_ID_UNIT_02.Text[28] := "M_ONE" AND "DB4000_FIX_TABLE_POSITIONS".UNIT_02.FIXTURE_1.IN_MEASURING_STATION_2;
   "DB7235_VARIABLE_LAYOUT".PART_ID_UNIT_02.Image[2] := "M_ONE" AND "DB4000_FIX_TABLE_POSITIONS".UNIT_02.FIXTURE_1.IN_CLADDING_STATION_3;
   "DB7235_VARIABLE_LAYOUT".PART_ID_UNIT_02.Text[29] := "M_ONE" AND "DB4000_FIX_TABLE_POSITIONS".UNIT_02.FIXTURE_1.IN_CLADDING_STATION_3;
   "DB7235_VARIABLE_LAYOUT".PART_ID_UNIT_02.Text[24] := "M_ONE" AND "DB4000_FIX_TABLE_POSITIONS".UNIT_02.FIXTURE_1.IN_CLADDING_STATION_3;
   "DB7235_VARIABLE_LAYOUT".PART_ID_UNIT_02.Text[22] := "M_ONE" AND "DB4000_FIX_TABLE_POSITIONS".UNIT_02.FIXTURE_1.IN_CLADDING_STATION_3;
   "DB7235_VARIABLE_LAYOUT".PART_ID_UNIT_02.Text[32] := "M_ONE" AND "DB4000_FIX_TABLE_POSITIONS".UNIT_02.FIXTURE_1.IN_CLADDING_STATION_3;
   "DB7235_VARIABLE_LAYOUT".PART_ID_UNIT_02.Image[3] := "M_ONE" AND "DB4000_FIX_TABLE_POSITIONS".UNIT_02.FIXTURE_1.IN_CLEAN_STATION_4;
   "DB7235_VARIABLE_LAYOUT".PART_ID_UNIT_02.Text[31] := "M_ONE" AND "DB4000_FIX_TABLE_POSITIONS".UNIT_02.FIXTURE_1.IN_CLEAN_STATION_4;
   "DB7235_VARIABLE_LAYOUT".PART_ID_UNIT_02.Text[27] := "M_ONE" AND "DB4000_FIX_TABLE_POSITIONS".UNIT_02.FIXTURE_1.IN_CLEAN_STATION_4;
   "DB7235_VARIABLE_LAYOUT".PART_ID_UNIT_02.Text[20] := "M_ONE" AND "DB4000_FIX_TABLE_POSITIONS".UNIT_02.FIXTURE_1.IN_CLEAN_STATION_4;
   "DB7235_VARIABLE_LAYOUT".PART_ID_UNIT_02.Text[23] := "M_ONE" AND "DB4000_FIX_TABLE_POSITIONS".UNIT_02.FIXTURE_1.IN_CLEAN_STATION_4;
   "DB7235_VARIABLE_LAYOUT".PART_ID_UNIT_02.Image[4] := "M_ONE" AND "DB4000_FIX_TABLE_POSITIONS".UNIT_02.AXIS_E20_NOT_DEFINED_POS AND NOT "LBP_Axis15".E_NactNmin;
END_REGION

REGION Network 19: PC STATUS UNIT 01
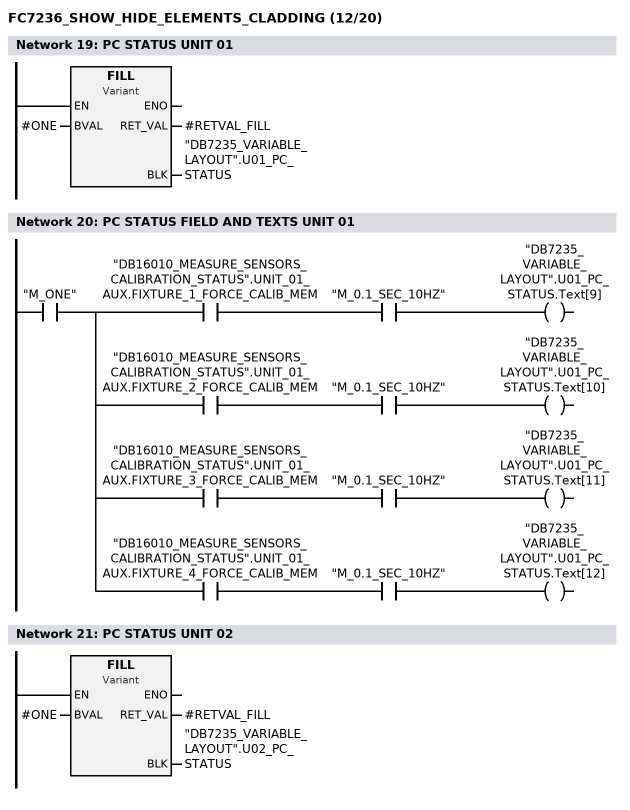
   RUNG wire#powerrail
      { S7_Templates := "ptr_type := Variant" } FILL(BVAL := #ONE, RET_VAL => #RETVAL_FILL, BLK => "DB7235_VARIABLE_LAYOUT".U01_PC_STATUS)
   END_RUNG
   // the same network as SCL:
   #RETVAL_FILL := FILL(BVAL := #ONE, BLK => "DB7235_VARIABLE_LAYOUT".U01_PC_STATUS);
END_REGION

REGION Network 20: PC STATUS FIELD AND TEXTS UNIT 01
   RUNG wire#powerrail
      Contact( "M_ONE" )
      wire#w1
      Contact( "DB16010_MEASURE_SENSORS_CALIBRATION_STATUS".UNIT_01_AUX.FIXTURE_1_FORCE_CALIB_MEM )
      Contact( "M_0.1_SEC_10HZ" )
      Coil( "DB7235_VARIABLE_LAYOUT".U01_PC_STATUS.Text[9] )
   END_RUNG
   RUNG wire#w1
      Contact( "DB16010_MEASURE_SENSORS_CALIBRATION_STATUS".UNIT_01_AUX.FIXTURE_2_FORCE_CALIB_MEM )
      Contact( "M_0.1_SEC_10HZ" )
      Coil( "DB7235_VARIABLE_LAYOUT".U01_PC_STATUS.Text[10] )
   END_RUNG
   RUNG wire#w1
      Contact( "DB16010_MEASURE_SENSORS_CALIBRATION_STATUS".UNIT_01_AUX.FIXTURE_3_FORCE_CALIB_MEM )
      Contact( "M_0.1_SEC_10HZ" )
      Coil( "DB7235_VARIABLE_LAYOUT".U01_PC_STATUS.Text[11] )
   END_RUNG
   RUNG wire#w1
      Contact( "DB16010_MEASURE_SENSORS_CALIBRATION_STATUS".UNIT_01_AUX.FIXTURE_4_FORCE_CALIB_MEM )
      Contact( "M_0.1_SEC_10HZ" )
      Coil( "DB7235_VARIABLE_LAYOUT".U01_PC_STATUS.Text[12] )
   END_RUNG
   // the same network as SCL:
   "DB7235_VARIABLE_LAYOUT".U01_PC_STATUS.Text[9] := "M_ONE" AND "DB16010_MEASURE_SENSORS_CALIBRATION_STATUS".UNIT_01_AUX.FIXTURE_1_FORCE_CALIB_MEM AND "M_0.1_SEC_10HZ";
   "DB7235_VARIABLE_LAYOUT".U01_PC_STATUS.Text[10] := "M_ONE" AND "DB16010_MEASURE_SENSORS_CALIBRATION_STATUS".UNIT_01_AUX.FIXTURE_2_FORCE_CALIB_MEM AND "M_0.1_SEC_10HZ";
   "DB7235_VARIABLE_LAYOUT".U01_PC_STATUS.Text[11] := "M_ONE" AND "DB16010_MEASURE_SENSORS_CALIBRATION_STATUS".UNIT_01_AUX.FIXTURE_3_FORCE_CALIB_MEM AND "M_0.1_SEC_10HZ";
   "DB7235_VARIABLE_LAYOUT".U01_PC_STATUS.Text[12] := "M_ONE" AND "DB16010_MEASURE_SENSORS_CALIBRATION_STATUS".UNIT_01_AUX.FIXTURE_4_FORCE_CALIB_MEM AND "M_0.1_SEC_10HZ";
END_REGION

REGION Network 21: PC STATUS UNIT 02
   RUNG wire#powerrail
      { S7_Templates := "ptr_type := Variant" } FILL(BVAL := #ONE, RET_VAL => #RETVAL_FILL, BLK => "DB7235_VARIABLE_LAYOUT".U02_PC_STATUS)
   END_RUNG
   // the same network as SCL:
   #RETVAL_FILL := FILL(BVAL := #ONE, BLK => "DB7235_VARIABLE_LAYOUT".U02_PC_STATUS);
END_REGION

REGION Network 22: PC STATUS FIELD AND TEXTS UNIT 03
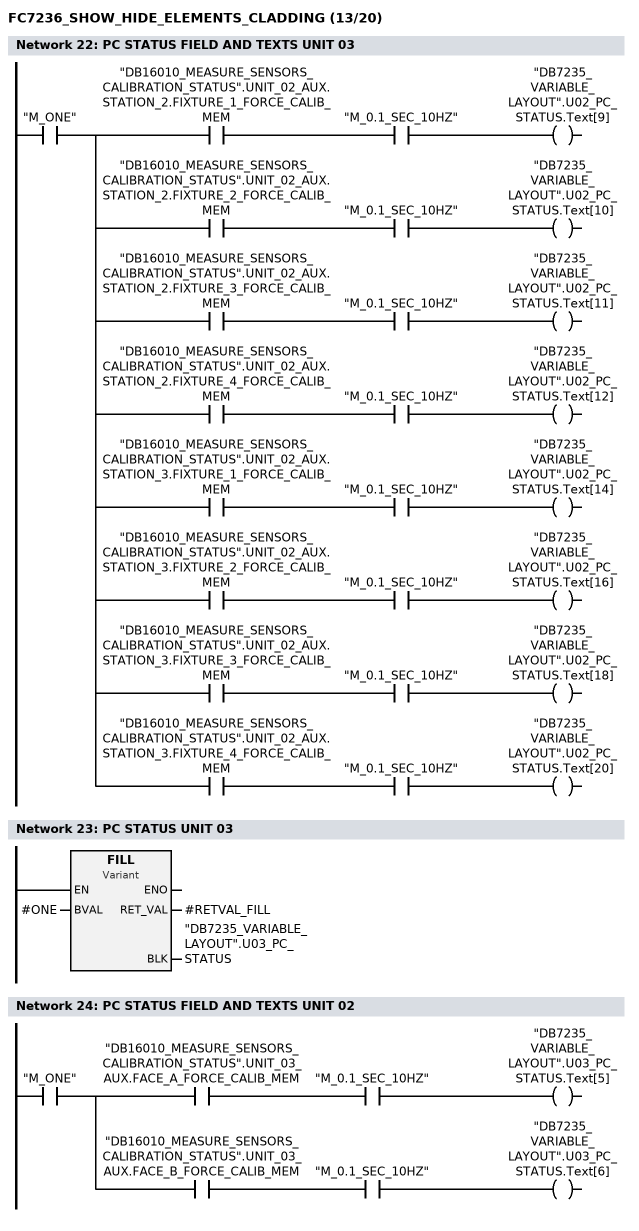
   RUNG wire#powerrail
      Contact( "M_ONE" )
      wire#w1
      Contact( "DB16010_MEASURE_SENSORS_CALIBRATION_STATUS".UNIT_02_AUX.STATION_2.FIXTURE_1_FORCE_CALIB_MEM )
      Contact( "M_0.1_SEC_10HZ" )
      Coil( "DB7235_VARIABLE_LAYOUT".U02_PC_STATUS.Text[9] )
   END_RUNG
   RUNG wire#w1
      Contact( "DB16010_MEASURE_SENSORS_CALIBRATION_STATUS".UNIT_02_AUX.STATION_2.FIXTURE_2_FORCE_CALIB_MEM )
      Contact( "M_0.1_SEC_10HZ" )
      Coil( "DB7235_VARIABLE_LAYOUT".U02_PC_STATUS.Text[10] )
   END_RUNG
   RUNG wire#w1
      Contact( "DB16010_MEASURE_SENSORS_CALIBRATION_STATUS".UNIT_02_AUX.STATION_2.FIXTURE_3_FORCE_CALIB_MEM )
      Contact( "M_0.1_SEC_10HZ" )
      Coil( "DB7235_VARIABLE_LAYOUT".U02_PC_STATUS.Text[11] )
   END_RUNG
   RUNG wire#w1
      Contact( "DB16010_MEASURE_SENSORS_CALIBRATION_STATUS".UNIT_02_AUX.STATION_2.FIXTURE_4_FORCE_CALIB_MEM )
      Contact( "M_0.1_SEC_10HZ" )
      Coil( "DB7235_VARIABLE_LAYOUT".U02_PC_STATUS.Text[12] )
   END_RUNG
   RUNG wire#w1
      Contact( "DB16010_MEASURE_SENSORS_CALIBRATION_STATUS".UNIT_02_AUX.STATION_3.FIXTURE_1_FORCE_CALIB_MEM )
      Contact( "M_0.1_SEC_10HZ" )
      Coil( "DB7235_VARIABLE_LAYOUT".U02_PC_STATUS.Text[14] )
   END_RUNG
   RUNG wire#w1
      Contact( "DB16010_MEASURE_SENSORS_CALIBRATION_STATUS".UNIT_02_AUX.STATION_3.FIXTURE_2_FORCE_CALIB_MEM )
      Contact( "M_0.1_SEC_10HZ" )
      Coil( "DB7235_VARIABLE_LAYOUT".U02_PC_STATUS.Text[16] )
   END_RUNG
   RUNG wire#w1
      Contact( "DB16010_MEASURE_SENSORS_CALIBRATION_STATUS".UNIT_02_AUX.STATION_3.FIXTURE_3_FORCE_CALIB_MEM )
      Contact( "M_0.1_SEC_10HZ" )
      Coil( "DB7235_VARIABLE_LAYOUT".U02_PC_STATUS.Text[18] )
   END_RUNG
   RUNG wire#w1
      Contact( "DB16010_MEASURE_SENSORS_CALIBRATION_STATUS".UNIT_02_AUX.STATION_3.FIXTURE_4_FORCE_CALIB_MEM )
      Contact( "M_0.1_SEC_10HZ" )
      Coil( "DB7235_VARIABLE_LAYOUT".U02_PC_STATUS.Text[20] )
   END_RUNG
   // the same network as SCL:
   "DB7235_VARIABLE_LAYOUT".U02_PC_STATUS.Text[9] := "M_ONE" AND "DB16010_MEASURE_SENSORS_CALIBRATION_STATUS".UNIT_02_AUX.STATION_2.FIXTURE_1_FORCE_CALIB_MEM AND "M_0.1_SEC_10HZ";
   "DB7235_VARIABLE_LAYOUT".U02_PC_STATUS.Text[10] := "M_ONE" AND "DB16010_MEASURE_SENSORS_CALIBRATION_STATUS".UNIT_02_AUX.STATION_2.FIXTURE_2_FORCE_CALIB_MEM AND "M_0.1_SEC_10HZ";
   "DB7235_VARIABLE_LAYOUT".U02_PC_STATUS.Text[11] := "M_ONE" AND "DB16010_MEASURE_SENSORS_CALIBRATION_STATUS".UNIT_02_AUX.STATION_2.FIXTURE_3_FORCE_CALIB_MEM AND "M_0.1_SEC_10HZ";
   "DB7235_VARIABLE_LAYOUT".U02_PC_STATUS.Text[12] := "M_ONE" AND "DB16010_MEASURE_SENSORS_CALIBRATION_STATUS".UNIT_02_AUX.STATION_2.FIXTURE_4_FORCE_CALIB_MEM AND "M_0.1_SEC_10HZ";
   "DB7235_VARIABLE_LAYOUT".U02_PC_STATUS.Text[14] := "M_ONE" AND "DB16010_MEASURE_SENSORS_CALIBRATION_STATUS".UNIT_02_AUX.STATION_3.FIXTURE_1_FORCE_CALIB_MEM AND "M_0.1_SEC_10HZ";
   "DB7235_VARIABLE_LAYOUT".U02_PC_STATUS.Text[16] := "M_ONE" AND "DB16010_MEASURE_SENSORS_CALIBRATION_STATUS".UNIT_02_AUX.STATION_3.FIXTURE_2_FORCE_CALIB_MEM AND "M_0.1_SEC_10HZ";
   "DB7235_VARIABLE_LAYOUT".U02_PC_STATUS.Text[18] := "M_ONE" AND "DB16010_MEASURE_SENSORS_CALIBRATION_STATUS".UNIT_02_AUX.STATION_3.FIXTURE_3_FORCE_CALIB_MEM AND "M_0.1_SEC_10HZ";
   "DB7235_VARIABLE_LAYOUT".U02_PC_STATUS.Text[20] := "M_ONE" AND "DB16010_MEASURE_SENSORS_CALIBRATION_STATUS".UNIT_02_AUX.STATION_3.FIXTURE_4_FORCE_CALIB_MEM AND "M_0.1_SEC_10HZ";
END_REGION

REGION Network 23: PC STATUS UNIT 03
   RUNG wire#powerrail
      { S7_Templates := "ptr_type := Variant" } FILL(BVAL := #ONE, RET_VAL => #RETVAL_FILL, BLK => "DB7235_VARIABLE_LAYOUT".U03_PC_STATUS)
   END_RUNG
   // the same network as SCL:
   #RETVAL_FILL := FILL(BVAL := #ONE, BLK => "DB7235_VARIABLE_LAYOUT".U03_PC_STATUS);
END_REGION

REGION Network 24: PC STATUS FIELD AND TEXTS UNIT 02
   RUNG wire#powerrail
      Contact( "M_ONE" )
      wire#w1
      Contact( "DB16010_MEASURE_SENSORS_CALIBRATION_STATUS".UNIT_03_AUX.FACE_A_FORCE_CALIB_MEM )
      Contact( "M_0.1_SEC_10HZ" )
      Coil( "DB7235_VARIABLE_LAYOUT".U03_PC_STATUS.Text[5] )
   END_RUNG
   RUNG wire#w1
      Contact( "DB16010_MEASURE_SENSORS_CALIBRATION_STATUS".UNIT_03_AUX.FACE_B_FORCE_CALIB_MEM )
      Contact( "M_0.1_SEC_10HZ" )
      Coil( "DB7235_VARIABLE_LAYOUT".U03_PC_STATUS.Text[6] )
   END_RUNG
   // the same network as SCL:
   "DB7235_VARIABLE_LAYOUT".U03_PC_STATUS.Text[5] := "M_ONE" AND "DB16010_MEASURE_SENSORS_CALIBRATION_STATUS".UNIT_03_AUX.FACE_A_FORCE_CALIB_MEM AND "M_0.1_SEC_10HZ";
   "DB7235_VARIABLE_LAYOUT".U03_PC_STATUS.Text[6] := "M_ONE" AND "DB16010_MEASURE_SENSORS_CALIBRATION_STATUS".UNIT_03_AUX.FACE_B_FORCE_CALIB_MEM AND "M_0.1_SEC_10HZ";
END_REGION

REGION Network 25: *************** ENABLE OR DISABLE ELEMENTS ***************
END_REGION

REGION Network 26: RFID
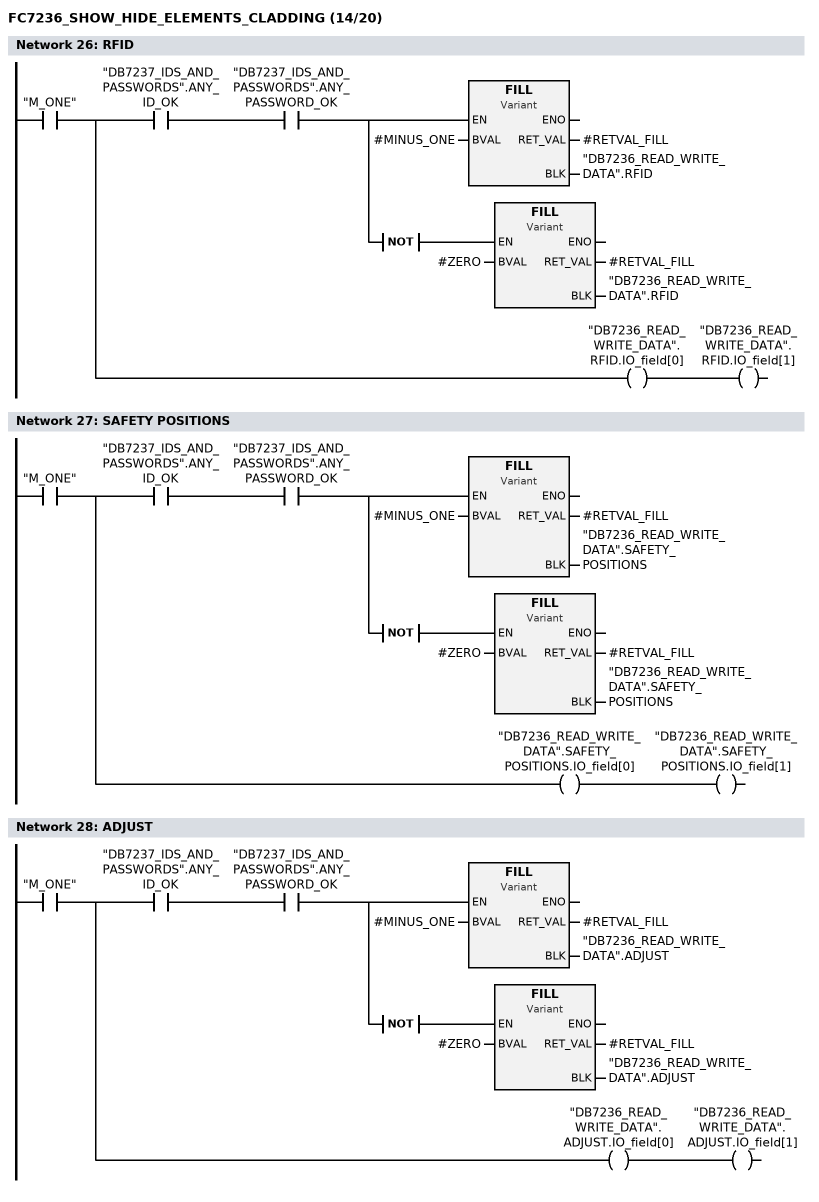
   RUNG wire#powerrail
      Contact( "M_ONE" )
      wire#w1
      Contact( "DB7237_IDS_AND_PASSWORDS".ANY_ID_OK )
      Contact( "DB7237_IDS_AND_PASSWORDS".ANY_PASSWORD_OK )
      wire#w2
      { S7_Templates := "ptr_type := Variant" } FILL(BVAL := #MINUS_ONE, RET_VAL => #RETVAL_FILL, BLK => "DB7236_READ_WRITE_DATA".RFID)
   END_RUNG
   RUNG wire#w2
      Not()
      { S7_Templates := "ptr_type := Variant" } FILL(BVAL := #ZERO, RET_VAL => #RETVAL_FILL, BLK => "DB7236_READ_WRITE_DATA".RFID)
   END_RUNG
   RUNG wire#w1
      Coil( "DB7236_READ_WRITE_DATA".RFID.IO_field[0] )
      Coil( "DB7236_READ_WRITE_DATA".RFID.IO_field[1] )
   END_RUNG
   // the same network as SCL:
   #_w1 := "M_ONE" AND "DB7237_IDS_AND_PASSWORDS".ANY_ID_OK AND "DB7237_IDS_AND_PASSWORDS".ANY_PASSWORD_OK;
   #_w2 := "M_ONE";
   IF #_w1 THEN #RETVAL_FILL := FILL(BVAL := #MINUS_ONE, BLK => "DB7236_READ_WRITE_DATA".RFID); END_IF;
   IF NOT #_w1 THEN #RETVAL_FILL := FILL(BVAL := #ZERO, BLK => "DB7236_READ_WRITE_DATA".RFID); END_IF;
   "DB7236_READ_WRITE_DATA".RFID.IO_field[0] := #_w2;
   "DB7236_READ_WRITE_DATA".RFID.IO_field[1] := #_w2;
END_REGION

REGION Network 27: SAFETY POSITIONS
   RUNG wire#powerrail
      Contact( "M_ONE" )
      wire#w1
      Contact( "DB7237_IDS_AND_PASSWORDS".ANY_ID_OK )
      Contact( "DB7237_IDS_AND_PASSWORDS".ANY_PASSWORD_OK )
      wire#w2
      { S7_Templates := "ptr_type := Variant" } FILL(BVAL := #MINUS_ONE, RET_VAL => #RETVAL_FILL, BLK => "DB7236_READ_WRITE_DATA".SAFETY_POSITIONS)
   END_RUNG
   RUNG wire#w2
      Not()
      { S7_Templates := "ptr_type := Variant" } FILL(BVAL := #ZERO, RET_VAL => #RETVAL_FILL, BLK => "DB7236_READ_WRITE_DATA".SAFETY_POSITIONS)
   END_RUNG
   RUNG wire#w1
      Coil( "DB7236_READ_WRITE_DATA".SAFETY_POSITIONS.IO_field[0] )
      Coil( "DB7236_READ_WRITE_DATA".SAFETY_POSITIONS.IO_field[1] )
   END_RUNG
   // the same network as SCL:
   #_w1 := "M_ONE" AND "DB7237_IDS_AND_PASSWORDS".ANY_ID_OK AND "DB7237_IDS_AND_PASSWORDS".ANY_PASSWORD_OK;
   #_w2 := "M_ONE";
   IF #_w1 THEN
       #RETVAL_FILL := FILL(BVAL := #MINUS_ONE, BLK => "DB7236_READ_WRITE_DATA".SAFETY_POSITIONS);
   END_IF;
   IF NOT #_w1 THEN
       #RETVAL_FILL := FILL(BVAL := #ZERO, BLK => "DB7236_READ_WRITE_DATA".SAFETY_POSITIONS);
   END_IF;
   "DB7236_READ_WRITE_DATA".SAFETY_POSITIONS.IO_field[0] := #_w2;
   "DB7236_READ_WRITE_DATA".SAFETY_POSITIONS.IO_field[1] := #_w2;
END_REGION

REGION Network 28: ADJUST
   RUNG wire#powerrail
      Contact( "M_ONE" )
      wire#w1
      Contact( "DB7237_IDS_AND_PASSWORDS".ANY_ID_OK )
      Contact( "DB7237_IDS_AND_PASSWORDS".ANY_PASSWORD_OK )
      wire#w2
      { S7_Templates := "ptr_type := Variant" } FILL(BVAL := #MINUS_ONE, RET_VAL => #RETVAL_FILL, BLK => "DB7236_READ_WRITE_DATA".ADJUST)
   END_RUNG
   RUNG wire#w2
      Not()
      { S7_Templates := "ptr_type := Variant" } FILL(BVAL := #ZERO, RET_VAL => #RETVAL_FILL, BLK => "DB7236_READ_WRITE_DATA".ADJUST)
   END_RUNG
   RUNG wire#w1
      Coil( "DB7236_READ_WRITE_DATA".ADJUST.IO_field[0] )
      Coil( "DB7236_READ_WRITE_DATA".ADJUST.IO_field[1] )
   END_RUNG
   // the same network as SCL:
   #_w1 := "M_ONE" AND "DB7237_IDS_AND_PASSWORDS".ANY_ID_OK AND "DB7237_IDS_AND_PASSWORDS".ANY_PASSWORD_OK;
   #_w2 := "M_ONE";
   IF #_w1 THEN #RETVAL_FILL := FILL(BVAL := #MINUS_ONE, BLK => "DB7236_READ_WRITE_DATA".ADJUST); END_IF;
   IF NOT #_w1 THEN #RETVAL_FILL := FILL(BVAL := #ZERO, BLK => "DB7236_READ_WRITE_DATA".ADJUST); END_IF;
   "DB7236_READ_WRITE_DATA".ADJUST.IO_field[0] := #_w2;
   "DB7236_READ_WRITE_DATA".ADJUST.IO_field[1] := #_w2;
END_REGION

REGION Network 29: ANALOGS
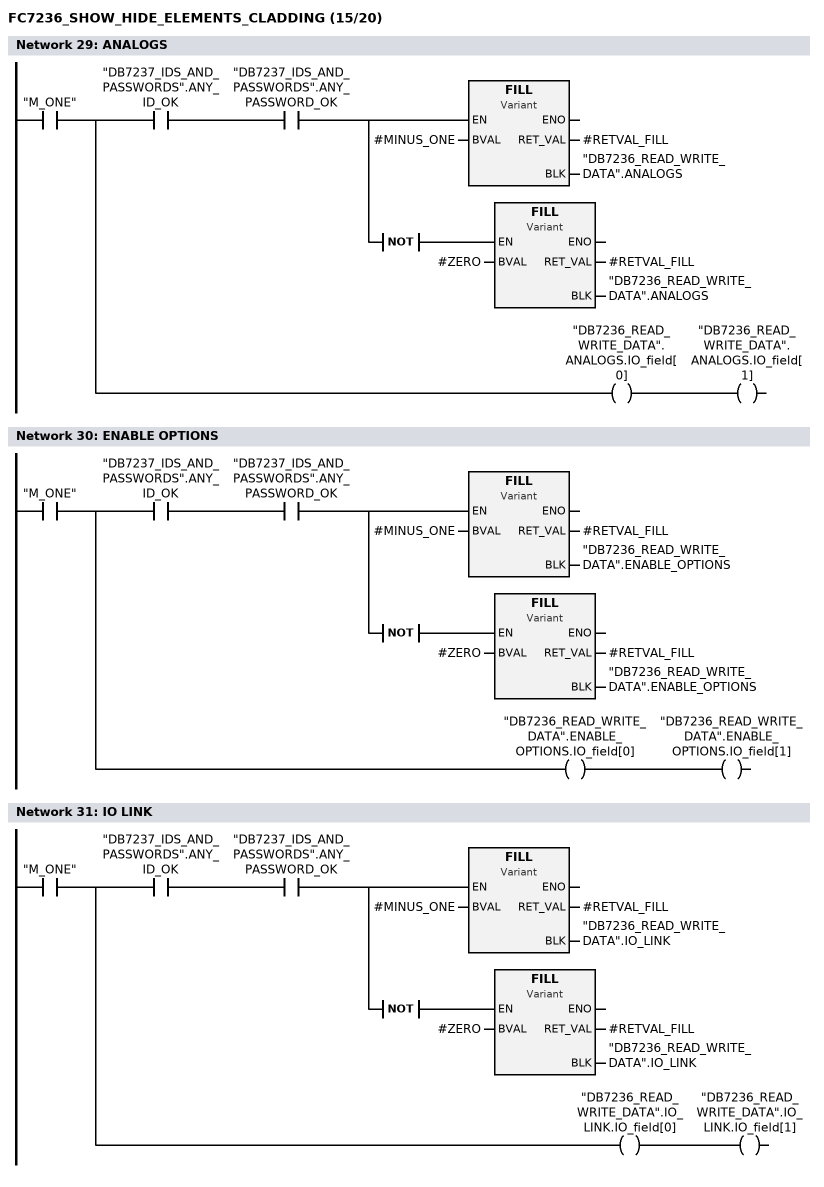
   RUNG wire#powerrail
      Contact( "M_ONE" )
      wire#w1
      Contact( "DB7237_IDS_AND_PASSWORDS".ANY_ID_OK )
      Contact( "DB7237_IDS_AND_PASSWORDS".ANY_PASSWORD_OK )
      wire#w2
      { S7_Templates := "ptr_type := Variant" } FILL(BVAL := #MINUS_ONE, RET_VAL => #RETVAL_FILL, BLK => "DB7236_READ_WRITE_DATA".ANALOGS)
   END_RUNG
   RUNG wire#w2
      Not()
      { S7_Templates := "ptr_type := Variant" } FILL(BVAL := #ZERO, RET_VAL => #RETVAL_FILL, BLK => "DB7236_READ_WRITE_DATA".ANALOGS)
   END_RUNG
   RUNG wire#w1
      Coil( "DB7236_READ_WRITE_DATA".ANALOGS.IO_field[0] )
      Coil( "DB7236_READ_WRITE_DATA".ANALOGS.IO_field[1] )
   END_RUNG
   // the same network as SCL:
   #_w1 := "M_ONE" AND "DB7237_IDS_AND_PASSWORDS".ANY_ID_OK AND "DB7237_IDS_AND_PASSWORDS".ANY_PASSWORD_OK;
   #_w2 := "M_ONE";
   IF #_w1 THEN #RETVAL_FILL := FILL(BVAL := #MINUS_ONE, BLK => "DB7236_READ_WRITE_DATA".ANALOGS); END_IF;
   IF NOT #_w1 THEN #RETVAL_FILL := FILL(BVAL := #ZERO, BLK => "DB7236_READ_WRITE_DATA".ANALOGS); END_IF;
   "DB7236_READ_WRITE_DATA".ANALOGS.IO_field[0] := #_w2;
   "DB7236_READ_WRITE_DATA".ANALOGS.IO_field[1] := #_w2;
END_REGION

REGION Network 30: ENABLE OPTIONS
   RUNG wire#powerrail
      Contact( "M_ONE" )
      wire#w1
      Contact( "DB7237_IDS_AND_PASSWORDS".ANY_ID_OK )
      Contact( "DB7237_IDS_AND_PASSWORDS".ANY_PASSWORD_OK )
      wire#w2
      { S7_Templates := "ptr_type := Variant" } FILL(BVAL := #MINUS_ONE, RET_VAL => #RETVAL_FILL, BLK => "DB7236_READ_WRITE_DATA".ENABLE_OPTIONS)
   END_RUNG
   RUNG wire#w2
      Not()
      { S7_Templates := "ptr_type := Variant" } FILL(BVAL := #ZERO, RET_VAL => #RETVAL_FILL, BLK => "DB7236_READ_WRITE_DATA".ENABLE_OPTIONS)
   END_RUNG
   RUNG wire#w1
      Coil( "DB7236_READ_WRITE_DATA".ENABLE_OPTIONS.IO_field[0] )
      Coil( "DB7236_READ_WRITE_DATA".ENABLE_OPTIONS.IO_field[1] )
   END_RUNG
   // the same network as SCL:
   #_w1 := "M_ONE" AND "DB7237_IDS_AND_PASSWORDS".ANY_ID_OK AND "DB7237_IDS_AND_PASSWORDS".ANY_PASSWORD_OK;
   #_w2 := "M_ONE";
   IF #_w1 THEN
       #RETVAL_FILL := FILL(BVAL := #MINUS_ONE, BLK => "DB7236_READ_WRITE_DATA".ENABLE_OPTIONS);
   END_IF;
   IF NOT #_w1 THEN
       #RETVAL_FILL := FILL(BVAL := #ZERO, BLK => "DB7236_READ_WRITE_DATA".ENABLE_OPTIONS);
   END_IF;
   "DB7236_READ_WRITE_DATA".ENABLE_OPTIONS.IO_field[0] := #_w2;
   "DB7236_READ_WRITE_DATA".ENABLE_OPTIONS.IO_field[1] := #_w2;
END_REGION

REGION Network 31: IO LINK
   RUNG wire#powerrail
      Contact( "M_ONE" )
      wire#w1
      Contact( "DB7237_IDS_AND_PASSWORDS".ANY_ID_OK )
      Contact( "DB7237_IDS_AND_PASSWORDS".ANY_PASSWORD_OK )
      wire#w2
      { S7_Templates := "ptr_type := Variant" } FILL(BVAL := #MINUS_ONE, RET_VAL => #RETVAL_FILL, BLK => "DB7236_READ_WRITE_DATA".IO_LINK)
   END_RUNG
   RUNG wire#w2
      Not()
      { S7_Templates := "ptr_type := Variant" } FILL(BVAL := #ZERO, RET_VAL => #RETVAL_FILL, BLK => "DB7236_READ_WRITE_DATA".IO_LINK)
   END_RUNG
   RUNG wire#w1
      Coil( "DB7236_READ_WRITE_DATA".IO_LINK.IO_field[0] )
      Coil( "DB7236_READ_WRITE_DATA".IO_LINK.IO_field[1] )
   END_RUNG
   // the same network as SCL:
   #_w1 := "M_ONE" AND "DB7237_IDS_AND_PASSWORDS".ANY_ID_OK AND "DB7237_IDS_AND_PASSWORDS".ANY_PASSWORD_OK;
   #_w2 := "M_ONE";
   IF #_w1 THEN #RETVAL_FILL := FILL(BVAL := #MINUS_ONE, BLK => "DB7236_READ_WRITE_DATA".IO_LINK); END_IF;
   IF NOT #_w1 THEN #RETVAL_FILL := FILL(BVAL := #ZERO, BLK => "DB7236_READ_WRITE_DATA".IO_LINK); END_IF;
   "DB7236_READ_WRITE_DATA".IO_LINK.IO_field[0] := #_w2;
   "DB7236_READ_WRITE_DATA".IO_LINK.IO_field[1] := #_w2;
END_REGION

REGION Network 32: MASS CENTER
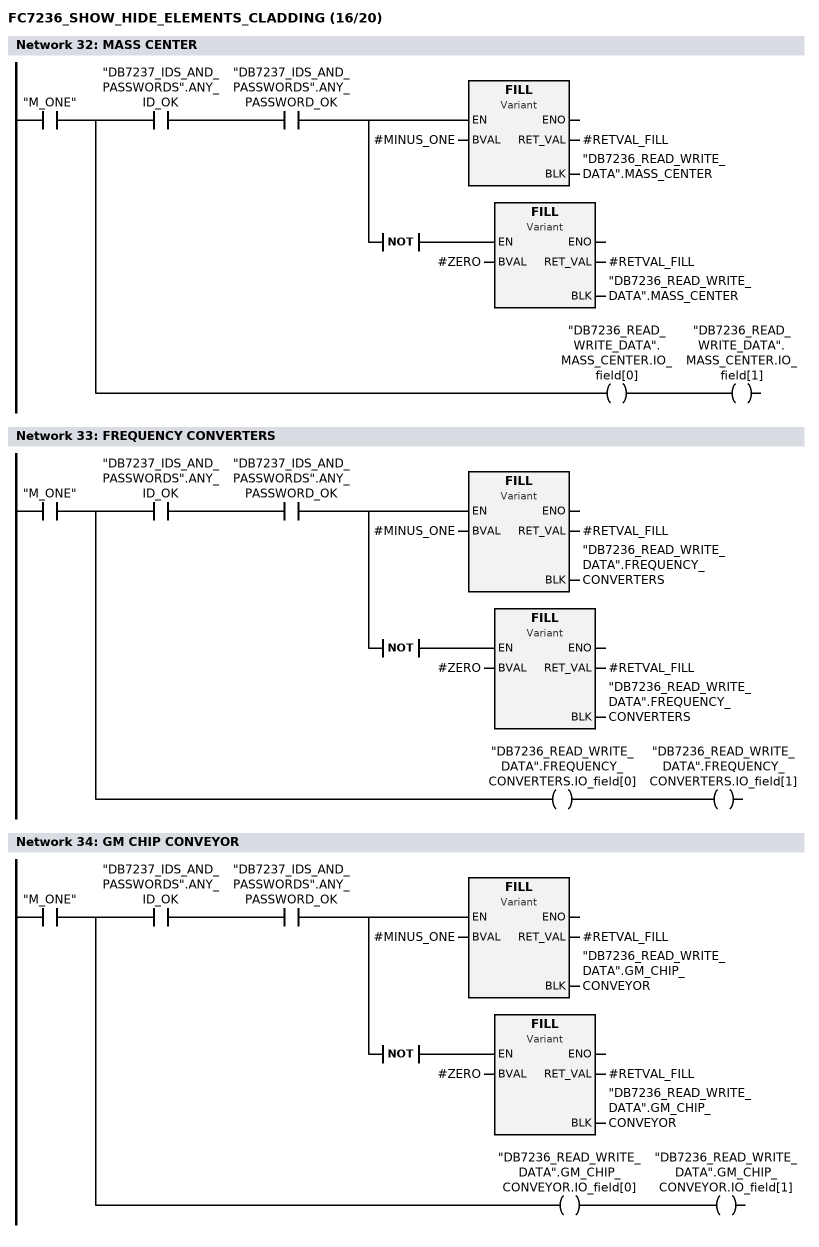
   RUNG wire#powerrail
      Contact( "M_ONE" )
      wire#w1
      Contact( "DB7237_IDS_AND_PASSWORDS".ANY_ID_OK )
      Contact( "DB7237_IDS_AND_PASSWORDS".ANY_PASSWORD_OK )
      wire#w2
      { S7_Templates := "ptr_type := Variant" } FILL(BVAL := #MINUS_ONE, RET_VAL => #RETVAL_FILL, BLK => "DB7236_READ_WRITE_DATA".MASS_CENTER)
   END_RUNG
   RUNG wire#w2
      Not()
      { S7_Templates := "ptr_type := Variant" } FILL(BVAL := #ZERO, RET_VAL => #RETVAL_FILL, BLK => "DB7236_READ_WRITE_DATA".MASS_CENTER)
   END_RUNG
   RUNG wire#w1
      Coil( "DB7236_READ_WRITE_DATA".MASS_CENTER.IO_field[0] )
      Coil( "DB7236_READ_WRITE_DATA".MASS_CENTER.IO_field[1] )
   END_RUNG
   // the same network as SCL:
   #_w1 := "M_ONE" AND "DB7237_IDS_AND_PASSWORDS".ANY_ID_OK AND "DB7237_IDS_AND_PASSWORDS".ANY_PASSWORD_OK;
   #_w2 := "M_ONE";
   IF #_w1 THEN
       #RETVAL_FILL := FILL(BVAL := #MINUS_ONE, BLK => "DB7236_READ_WRITE_DATA".MASS_CENTER);
   END_IF;
   IF NOT #_w1 THEN #RETVAL_FILL := FILL(BVAL := #ZERO, BLK => "DB7236_READ_WRITE_DATA".MASS_CENTER); END_IF;
   "DB7236_READ_WRITE_DATA".MASS_CENTER.IO_field[0] := #_w2;
   "DB7236_READ_WRITE_DATA".MASS_CENTER.IO_field[1] := #_w2;
END_REGION

REGION Network 33: FREQUENCY CONVERTERS
   RUNG wire#powerrail
      Contact( "M_ONE" )
      wire#w1
      Contact( "DB7237_IDS_AND_PASSWORDS".ANY_ID_OK )
      Contact( "DB7237_IDS_AND_PASSWORDS".ANY_PASSWORD_OK )
      wire#w2
      { S7_Templates := "ptr_type := Variant" } FILL(BVAL := #MINUS_ONE, RET_VAL => #RETVAL_FILL, BLK => "DB7236_READ_WRITE_DATA".FREQUENCY_CONVERTERS)
   END_RUNG
   RUNG wire#w2
      Not()
      { S7_Templates := "ptr_type := Variant" } FILL(BVAL := #ZERO, RET_VAL => #RETVAL_FILL, BLK => "DB7236_READ_WRITE_DATA".FREQUENCY_CONVERTERS)
   END_RUNG
   RUNG wire#w1
      Coil( "DB7236_READ_WRITE_DATA".FREQUENCY_CONVERTERS.IO_field[0] )
      Coil( "DB7236_READ_WRITE_DATA".FREQUENCY_CONVERTERS.IO_field[1] )
   END_RUNG
   // the same network as SCL:
   #_w1 := "M_ONE" AND "DB7237_IDS_AND_PASSWORDS".ANY_ID_OK AND "DB7237_IDS_AND_PASSWORDS".ANY_PASSWORD_OK;
   #_w2 := "M_ONE";
   IF #_w1 THEN
       #RETVAL_FILL := FILL(BVAL := #MINUS_ONE, BLK => "DB7236_READ_WRITE_DATA".FREQUENCY_CONVERTERS);
   END_IF;
   IF NOT #_w1 THEN
       #RETVAL_FILL := FILL(BVAL := #ZERO, BLK => "DB7236_READ_WRITE_DATA".FREQUENCY_CONVERTERS);
   END_IF;
   "DB7236_READ_WRITE_DATA".FREQUENCY_CONVERTERS.IO_field[0] := #_w2;
   "DB7236_READ_WRITE_DATA".FREQUENCY_CONVERTERS.IO_field[1] := #_w2;
END_REGION

REGION Network 34: GM CHIP CONVEYOR
   RUNG wire#powerrail
      Contact( "M_ONE" )
      wire#w1
      Contact( "DB7237_IDS_AND_PASSWORDS".ANY_ID_OK )
      Contact( "DB7237_IDS_AND_PASSWORDS".ANY_PASSWORD_OK )
      wire#w2
      { S7_Templates := "ptr_type := Variant" } FILL(BVAL := #MINUS_ONE, RET_VAL => #RETVAL_FILL, BLK => "DB7236_READ_WRITE_DATA".GM_CHIP_CONVEYOR)
   END_RUNG
   RUNG wire#w2
      Not()
      { S7_Templates := "ptr_type := Variant" } FILL(BVAL := #ZERO, RET_VAL => #RETVAL_FILL, BLK => "DB7236_READ_WRITE_DATA".GM_CHIP_CONVEYOR)
   END_RUNG
   RUNG wire#w1
      Coil( "DB7236_READ_WRITE_DATA".GM_CHIP_CONVEYOR.IO_field[0] )
      Coil( "DB7236_READ_WRITE_DATA".GM_CHIP_CONVEYOR.IO_field[1] )
   END_RUNG
   // the same network as SCL:
   #_w1 := "M_ONE" AND "DB7237_IDS_AND_PASSWORDS".ANY_ID_OK AND "DB7237_IDS_AND_PASSWORDS".ANY_PASSWORD_OK;
   #_w2 := "M_ONE";
   IF #_w1 THEN
       #RETVAL_FILL := FILL(BVAL := #MINUS_ONE, BLK => "DB7236_READ_WRITE_DATA".GM_CHIP_CONVEYOR);
   END_IF;
   IF NOT #_w1 THEN
       #RETVAL_FILL := FILL(BVAL := #ZERO, BLK => "DB7236_READ_WRITE_DATA".GM_CHIP_CONVEYOR);
   END_IF;
   "DB7236_READ_WRITE_DATA".GM_CHIP_CONVEYOR.IO_field[0] := #_w2;
   "DB7236_READ_WRITE_DATA".GM_CHIP_CONVEYOR.IO_field[1] := #_w2;
END_REGION

REGION Network 35: BK MIKRO
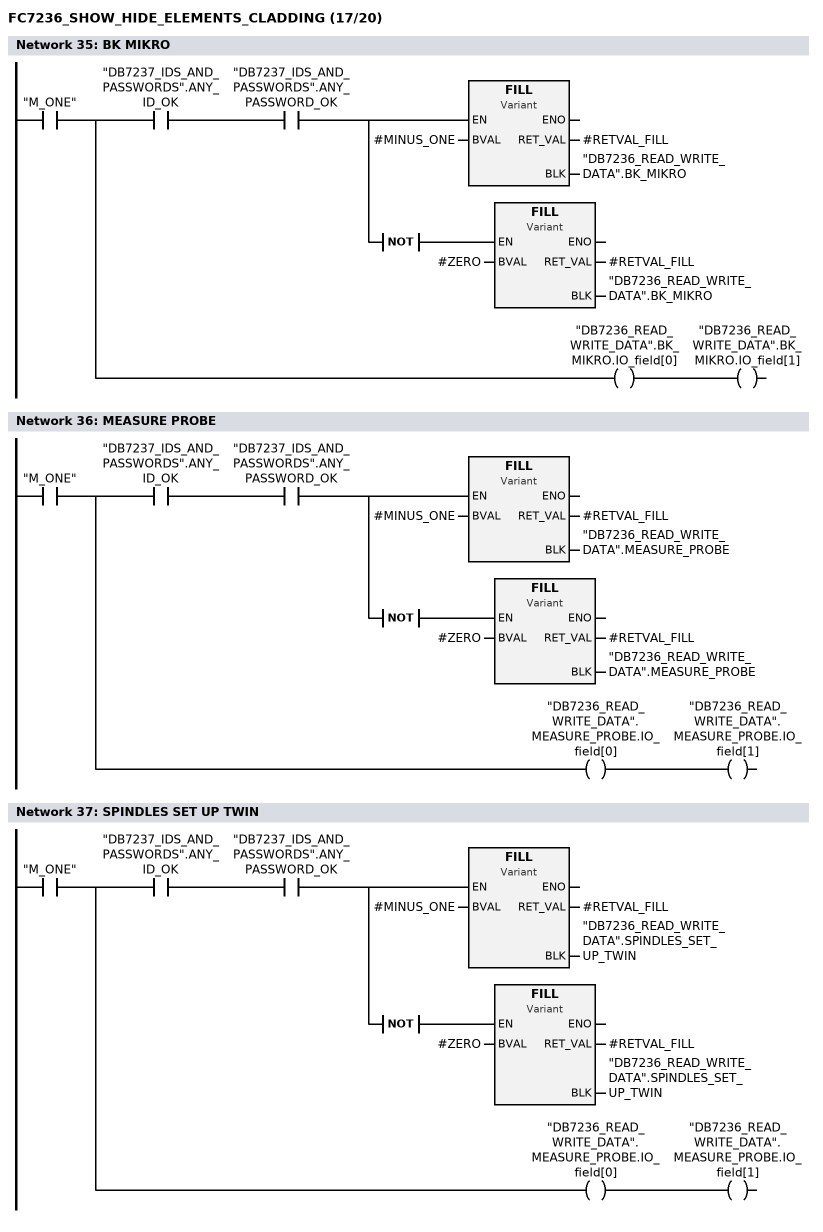
   RUNG wire#powerrail
      Contact( "M_ONE" )
      wire#w1
      Contact( "DB7237_IDS_AND_PASSWORDS".ANY_ID_OK )
      Contact( "DB7237_IDS_AND_PASSWORDS".ANY_PASSWORD_OK )
      wire#w2
      { S7_Templates := "ptr_type := Variant" } FILL(BVAL := #MINUS_ONE, RET_VAL => #RETVAL_FILL, BLK => "DB7236_READ_WRITE_DATA".BK_MIKRO)
   END_RUNG
   RUNG wire#w2
      Not()
      { S7_Templates := "ptr_type := Variant" } FILL(BVAL := #ZERO, RET_VAL => #RETVAL_FILL, BLK => "DB7236_READ_WRITE_DATA".BK_MIKRO)
   END_RUNG
   RUNG wire#w1
      Coil( "DB7236_READ_WRITE_DATA".BK_MIKRO.IO_field[0] )
      Coil( "DB7236_READ_WRITE_DATA".BK_MIKRO.IO_field[1] )
   END_RUNG
   // the same network as SCL:
   #_w1 := "M_ONE" AND "DB7237_IDS_AND_PASSWORDS".ANY_ID_OK AND "DB7237_IDS_AND_PASSWORDS".ANY_PASSWORD_OK;
   #_w2 := "M_ONE";
   IF #_w1 THEN #RETVAL_FILL := FILL(BVAL := #MINUS_ONE, BLK => "DB7236_READ_WRITE_DATA".BK_MIKRO); END_IF;
   IF NOT #_w1 THEN #RETVAL_FILL := FILL(BVAL := #ZERO, BLK => "DB7236_READ_WRITE_DATA".BK_MIKRO); END_IF;
   "DB7236_READ_WRITE_DATA".BK_MIKRO.IO_field[0] := #_w2;
   "DB7236_READ_WRITE_DATA".BK_MIKRO.IO_field[1] := #_w2;
END_REGION

REGION Network 36: MEASURE PROBE
   RUNG wire#powerrail
      Contact( "M_ONE" )
      wire#w1
      Contact( "DB7237_IDS_AND_PASSWORDS".ANY_ID_OK )
      Contact( "DB7237_IDS_AND_PASSWORDS".ANY_PASSWORD_OK )
      wire#w2
      { S7_Templates := "ptr_type := Variant" } FILL(BVAL := #MINUS_ONE, RET_VAL => #RETVAL_FILL, BLK => "DB7236_READ_WRITE_DATA".MEASURE_PROBE)
   END_RUNG
   RUNG wire#w2
      Not()
      { S7_Templates := "ptr_type := Variant" } FILL(BVAL := #ZERO, RET_VAL => #RETVAL_FILL, BLK => "DB7236_READ_WRITE_DATA".MEASURE_PROBE)
   END_RUNG
   RUNG wire#w1
      Coil( "DB7236_READ_WRITE_DATA".MEASURE_PROBE.IO_field[0] )
      Coil( "DB7236_READ_WRITE_DATA".MEASURE_PROBE.IO_field[1] )
   END_RUNG
   // the same network as SCL:
   #_w1 := "M_ONE" AND "DB7237_IDS_AND_PASSWORDS".ANY_ID_OK AND "DB7237_IDS_AND_PASSWORDS".ANY_PASSWORD_OK;
   #_w2 := "M_ONE";
   IF #_w1 THEN
       #RETVAL_FILL := FILL(BVAL := #MINUS_ONE, BLK => "DB7236_READ_WRITE_DATA".MEASURE_PROBE);
   END_IF;
   IF NOT #_w1 THEN
       #RETVAL_FILL := FILL(BVAL := #ZERO, BLK => "DB7236_READ_WRITE_DATA".MEASURE_PROBE);
   END_IF;
   "DB7236_READ_WRITE_DATA".MEASURE_PROBE.IO_field[0] := #_w2;
   "DB7236_READ_WRITE_DATA".MEASURE_PROBE.IO_field[1] := #_w2;
END_REGION

REGION Network 37: SPINDLES SET UP TWIN
   RUNG wire#powerrail
      Contact( "M_ONE" )
      wire#w1
      Contact( "DB7237_IDS_AND_PASSWORDS".ANY_ID_OK )
      Contact( "DB7237_IDS_AND_PASSWORDS".ANY_PASSWORD_OK )
      wire#w2
      { S7_Templates := "ptr_type := Variant" } FILL(BVAL := #MINUS_ONE, RET_VAL => #RETVAL_FILL, BLK => "DB7236_READ_WRITE_DATA".SPINDLES_SET_UP_TWIN)
   END_RUNG
   RUNG wire#w2
      Not()
      { S7_Templates := "ptr_type := Variant" } FILL(BVAL := #ZERO, RET_VAL => #RETVAL_FILL, BLK => "DB7236_READ_WRITE_DATA".SPINDLES_SET_UP_TWIN)
   END_RUNG
   RUNG wire#w1
      Coil( "DB7236_READ_WRITE_DATA".MEASURE_PROBE.IO_field[0] )
      Coil( "DB7236_READ_WRITE_DATA".MEASURE_PROBE.IO_field[1] )
   END_RUNG
   // the same network as SCL:
   #_w1 := "M_ONE" AND "DB7237_IDS_AND_PASSWORDS".ANY_ID_OK AND "DB7237_IDS_AND_PASSWORDS".ANY_PASSWORD_OK;
   #_w2 := "M_ONE";
   IF #_w1 THEN
       #RETVAL_FILL := FILL(BVAL := #MINUS_ONE, BLK => "DB7236_READ_WRITE_DATA".SPINDLES_SET_UP_TWIN);
   END_IF;
   IF NOT #_w1 THEN
       #RETVAL_FILL := FILL(BVAL := #ZERO, BLK => "DB7236_READ_WRITE_DATA".SPINDLES_SET_UP_TWIN);
   END_IF;
   "DB7236_READ_WRITE_DATA".MEASURE_PROBE.IO_field[0] := #_w2;
   "DB7236_READ_WRITE_DATA".MEASURE_PROBE.IO_field[1] := #_w2;
END_REGION

REGION Network 38: ETXETAR
   // ONLY FOR ETXETAR USE
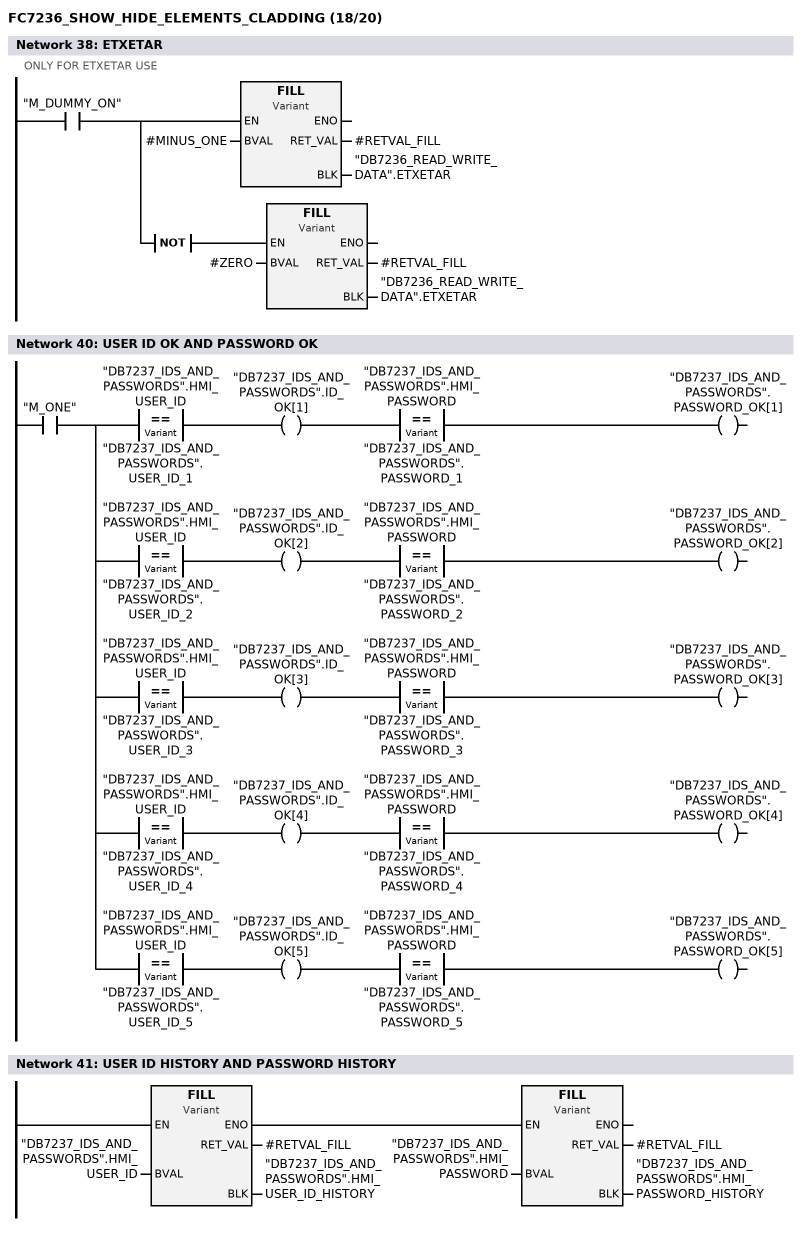
   RUNG wire#powerrail
      Contact( "M_DUMMY_ON" )
      wire#w1
      { S7_Templates := "ptr_type := Variant" } FILL(BVAL := #MINUS_ONE, RET_VAL => #RETVAL_FILL, BLK => "DB7236_READ_WRITE_DATA".ETXETAR)
   END_RUNG
   RUNG wire#w1
      Not()
      { S7_Templates := "ptr_type := Variant" } FILL(BVAL := #ZERO, RET_VAL => #RETVAL_FILL, BLK => "DB7236_READ_WRITE_DATA".ETXETAR)
   END_RUNG
   // the same network as SCL:
   #_w1 := "M_DUMMY_ON";
   IF #_w1 THEN #RETVAL_FILL := FILL(BVAL := #MINUS_ONE, BLK => "DB7236_READ_WRITE_DATA".ETXETAR); END_IF;
   IF NOT #_w1 THEN #RETVAL_FILL := FILL(BVAL := #ZERO, BLK => "DB7236_READ_WRITE_DATA".ETXETAR); END_IF;
END_REGION

REGION Network 39: **********************************************************
END_REGION

REGION Network 40: USER ID OK AND PASSWORD OK
   RUNG wire#powerrail
      Contact( "M_ONE" )
      wire#w1
      { S7_Templates := "SrcType := Variant" } EQ_Contact(in1 := "DB7237_IDS_AND_PASSWORDS".HMI_USER_ID, in2 := "DB7237_IDS_AND_PASSWORDS".USER_ID_1)
      Coil( "DB7237_IDS_AND_PASSWORDS".ID_OK[1] )
      { S7_Templates := "SrcType := Variant" } EQ_Contact(in1 := "DB7237_IDS_AND_PASSWORDS".HMI_PASSWORD, in2 := "DB7237_IDS_AND_PASSWORDS".PASSWORD_1)
      Coil( "DB7237_IDS_AND_PASSWORDS".PASSWORD_OK[1] )
   END_RUNG
   RUNG wire#w1
      { S7_Templates := "SrcType := Variant" } EQ_Contact(in1 := "DB7237_IDS_AND_PASSWORDS".HMI_USER_ID, in2 := "DB7237_IDS_AND_PASSWORDS".USER_ID_2)
      Coil( "DB7237_IDS_AND_PASSWORDS".ID_OK[2] )
      { S7_Templates := "SrcType := Variant" } EQ_Contact(in1 := "DB7237_IDS_AND_PASSWORDS".HMI_PASSWORD, in2 := "DB7237_IDS_AND_PASSWORDS".PASSWORD_2)
      Coil( "DB7237_IDS_AND_PASSWORDS".PASSWORD_OK[2] )
   END_RUNG
   RUNG wire#w1
      { S7_Templates := "SrcType := Variant" } EQ_Contact(in1 := "DB7237_IDS_AND_PASSWORDS".HMI_USER_ID, in2 := "DB7237_IDS_AND_PASSWORDS".USER_ID_3)
      Coil( "DB7237_IDS_AND_PASSWORDS".ID_OK[3] )
      { S7_Templates := "SrcType := Variant" } EQ_Contact(in1 := "DB7237_IDS_AND_PASSWORDS".HMI_PASSWORD, in2 := "DB7237_IDS_AND_PASSWORDS".PASSWORD_3)
      Coil( "DB7237_IDS_AND_PASSWORDS".PASSWORD_OK[3] )
   END_RUNG
   RUNG wire#w1
      { S7_Templates := "SrcType := Variant" } EQ_Contact(in1 := "DB7237_IDS_AND_PASSWORDS".HMI_USER_ID, in2 := "DB7237_IDS_AND_PASSWORDS".USER_ID_4)
      Coil( "DB7237_IDS_AND_PASSWORDS".ID_OK[4] )
      { S7_Templates := "SrcType := Variant" } EQ_Contact(in1 := "DB7237_IDS_AND_PASSWORDS".HMI_PASSWORD, in2 := "DB7237_IDS_AND_PASSWORDS".PASSWORD_4)
      Coil( "DB7237_IDS_AND_PASSWORDS".PASSWORD_OK[4] )
   END_RUNG
   RUNG wire#w1
      { S7_Templates := "SrcType := Variant" } EQ_Contact(in1 := "DB7237_IDS_AND_PASSWORDS".HMI_USER_ID, in2 := "DB7237_IDS_AND_PASSWORDS".USER_ID_5)
      Coil( "DB7237_IDS_AND_PASSWORDS".ID_OK[5] )
      { S7_Templates := "SrcType := Variant" } EQ_Contact(in1 := "DB7237_IDS_AND_PASSWORDS".HMI_PASSWORD, in2 := "DB7237_IDS_AND_PASSWORDS".PASSWORD_5)
      Coil( "DB7237_IDS_AND_PASSWORDS".PASSWORD_OK[5] )
   END_RUNG
   // the same network as SCL:
   "DB7237_IDS_AND_PASSWORDS".ID_OK[1] := "M_ONE" AND ("DB7237_IDS_AND_PASSWORDS".HMI_USER_ID = "DB7237_IDS_AND_PASSWORDS".USER_ID_1);
   "DB7237_IDS_AND_PASSWORDS".PASSWORD_OK[1] := "M_ONE" AND ("DB7237_IDS_AND_PASSWORDS".HMI_USER_ID = "DB7237_IDS_AND_PASSWORDS".USER_ID_1) AND ("DB7237_IDS_AND_PASSWORDS".HMI_PASSWORD = "DB7237_IDS_AND_PASSWORDS".PASSWORD_1);
   "DB7237_IDS_AND_PASSWORDS".ID_OK[2] := "M_ONE" AND ("DB7237_IDS_AND_PASSWORDS".HMI_USER_ID = "DB7237_IDS_AND_PASSWORDS".USER_ID_2);
   "DB7237_IDS_AND_PASSWORDS".PASSWORD_OK[2] := "M_ONE" AND ("DB7237_IDS_AND_PASSWORDS".HMI_USER_ID = "DB7237_IDS_AND_PASSWORDS".USER_ID_2) AND ("DB7237_IDS_AND_PASSWORDS".HMI_PASSWORD = "DB7237_IDS_AND_PASSWORDS".PASSWORD_2);
   "DB7237_IDS_AND_PASSWORDS".ID_OK[3] := "M_ONE" AND ("DB7237_IDS_AND_PASSWORDS".HMI_USER_ID = "DB7237_IDS_AND_PASSWORDS".USER_ID_3);
   "DB7237_IDS_AND_PASSWORDS".PASSWORD_OK[3] := "M_ONE" AND ("DB7237_IDS_AND_PASSWORDS".HMI_USER_ID = "DB7237_IDS_AND_PASSWORDS".USER_ID_3) AND ("DB7237_IDS_AND_PASSWORDS".HMI_PASSWORD = "DB7237_IDS_AND_PASSWORDS".PASSWORD_3);
   "DB7237_IDS_AND_PASSWORDS".ID_OK[4] := "M_ONE" AND ("DB7237_IDS_AND_PASSWORDS".HMI_USER_ID = "DB7237_IDS_AND_PASSWORDS".USER_ID_4);
   "DB7237_IDS_AND_PASSWORDS".PASSWORD_OK[4] := "M_ONE" AND ("DB7237_IDS_AND_PASSWORDS".HMI_USER_ID = "DB7237_IDS_AND_PASSWORDS".USER_ID_4) AND ("DB7237_IDS_AND_PASSWORDS".HMI_PASSWORD = "DB7237_IDS_AND_PASSWORDS".PASSWORD_4);
   "DB7237_IDS_AND_PASSWORDS".ID_OK[5] := "M_ONE" AND ("DB7237_IDS_AND_PASSWORDS".HMI_USER_ID = "DB7237_IDS_AND_PASSWORDS".USER_ID_5);
   "DB7237_IDS_AND_PASSWORDS".PASSWORD_OK[5] := "M_ONE" AND ("DB7237_IDS_AND_PASSWORDS".HMI_USER_ID = "DB7237_IDS_AND_PASSWORDS".USER_ID_5) AND ("DB7237_IDS_AND_PASSWORDS".HMI_PASSWORD = "DB7237_IDS_AND_PASSWORDS".PASSWORD_5);
END_REGION

REGION Network 41: USER ID HISTORY AND PASSWORD HISTORY
   RUNG wire#powerrail
      { S7_Templates := "ptr_type := Variant" } FILL(BVAL := "DB7237_IDS_AND_PASSWORDS".HMI_USER_ID, RET_VAL => #RETVAL_FILL, BLK => "DB7237_IDS_AND_PASSWORDS".HMI_USER_ID_HISTORY)
      { S7_Templates := "ptr_type := Variant" } FILL(BVAL := "DB7237_IDS_AND_PASSWORDS".HMI_PASSWORD, RET_VAL => #RETVAL_FILL, BLK => "DB7237_IDS_AND_PASSWORDS".HMI_PASSWORD_HISTORY)
   END_RUNG
   // the same network as SCL:
   #RETVAL_FILL := FILL(BVAL := "DB7237_IDS_AND_PASSWORDS".HMI_USER_ID,
                        BLK => "DB7237_IDS_AND_PASSWORDS".HMI_USER_ID_HISTORY,
                        ENO => #_w1);
   IF #_w1 THEN
       #RETVAL_FILL := FILL(BVAL := "DB7237_IDS_AND_PASSWORDS".HMI_PASSWORD,
                            BLK => "DB7237_IDS_AND_PASSWORDS".HMI_PASSWORD_HISTORY);
   END_IF;
END_REGION

REGION Network 42: RESET ANY USER ID OK AND ANY PASSWORD OK
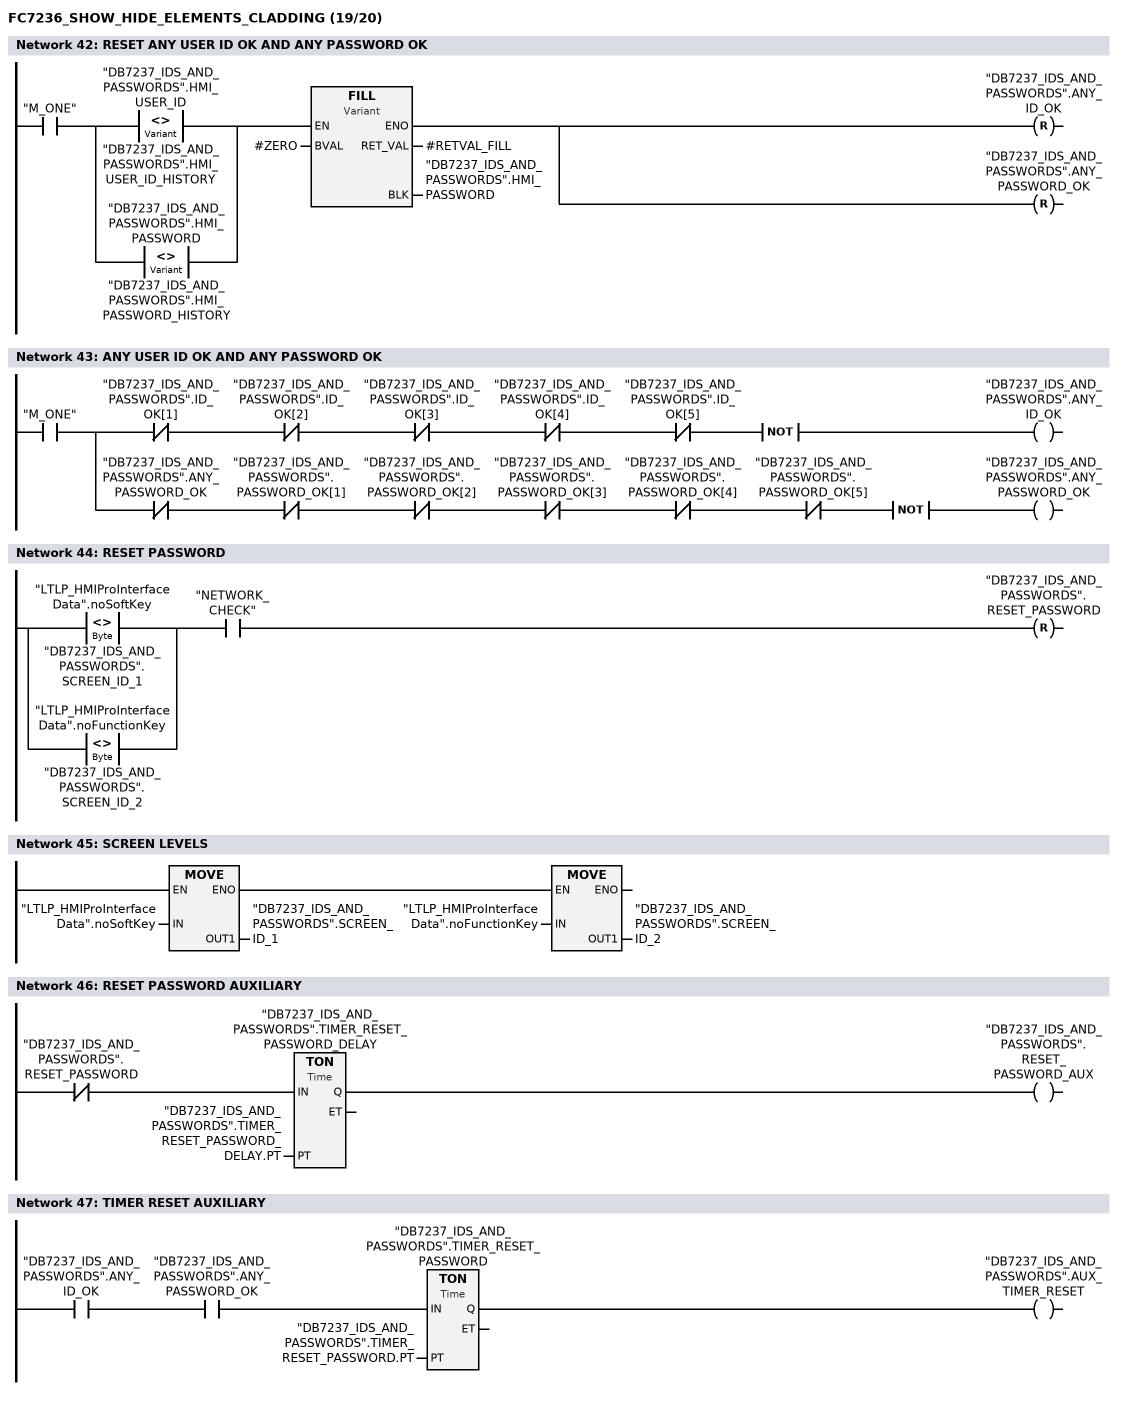
   RUNG wire#powerrail
      Contact( "M_ONE" )
      wire#w1
      { S7_Templates := "SrcType := Variant" } NE_Contact(in1 := "DB7237_IDS_AND_PASSWORDS".HMI_USER_ID, in2 := "DB7237_IDS_AND_PASSWORDS".HMI_USER_ID_HISTORY)
      wire#w2
      { S7_Templates := "ptr_type := Variant" } FILL(BVAL := #ZERO, RET_VAL => #RETVAL_FILL, BLK => "DB7237_IDS_AND_PASSWORDS".HMI_PASSWORD)
      wire#w3
      R_Coil( "DB7237_IDS_AND_PASSWORDS".ANY_ID_OK )
   END_RUNG
   RUNG wire#w1
      { S7_Templates := "SrcType := Variant" } NE_Contact(in1 := "DB7237_IDS_AND_PASSWORDS".HMI_PASSWORD, in2 := "DB7237_IDS_AND_PASSWORDS".HMI_PASSWORD_HISTORY)
   END_RUNG wire#w2
   RUNG wire#w3
      R_Coil( "DB7237_IDS_AND_PASSWORDS".ANY_PASSWORD_OK )
   END_RUNG
   // the same network as SCL:
   #RETVAL_FILL := FILL(EN := "M_ONE" AND (("DB7237_IDS_AND_PASSWORDS".HMI_USER_ID <> "DB7237_IDS_AND_PASSWORDS".HMI_USER_ID_HISTORY) OR ("DB7237_IDS_AND_PASSWORDS".HMI_PASSWORD <> "DB7237_IDS_AND_PASSWORDS".HMI_PASSWORD_HISTORY)),
                        BVAL := #ZERO,
                        BLK => "DB7237_IDS_AND_PASSWORDS".HMI_PASSWORD,
                        ENO => #_w1);
   IF #_w1 THEN
       "DB7237_IDS_AND_PASSWORDS".ANY_ID_OK := FALSE;
       "DB7237_IDS_AND_PASSWORDS".ANY_PASSWORD_OK := FALSE;
   END_IF;
END_REGION

REGION Network 43: ANY USER ID OK AND ANY PASSWORD OK
   RUNG wire#powerrail
      Contact( "M_ONE" )
      wire#w1
      I_Contact( "DB7237_IDS_AND_PASSWORDS".ID_OK[1] )
      I_Contact( "DB7237_IDS_AND_PASSWORDS".ID_OK[2] )
      I_Contact( "DB7237_IDS_AND_PASSWORDS".ID_OK[3] )
      I_Contact( "DB7237_IDS_AND_PASSWORDS".ID_OK[4] )
      I_Contact( "DB7237_IDS_AND_PASSWORDS".ID_OK[5] )
      Not()
      Coil( "DB7237_IDS_AND_PASSWORDS".ANY_ID_OK )
   END_RUNG
   RUNG wire#w1
      I_Contact( "DB7237_IDS_AND_PASSWORDS".ANY_PASSWORD_OK )
      I_Contact( "DB7237_IDS_AND_PASSWORDS".PASSWORD_OK[1] )
      I_Contact( "DB7237_IDS_AND_PASSWORDS".PASSWORD_OK[2] )
      I_Contact( "DB7237_IDS_AND_PASSWORDS".PASSWORD_OK[3] )
      I_Contact( "DB7237_IDS_AND_PASSWORDS".PASSWORD_OK[4] )
      I_Contact( "DB7237_IDS_AND_PASSWORDS".PASSWORD_OK[5] )
      Not()
      Coil( "DB7237_IDS_AND_PASSWORDS".ANY_PASSWORD_OK )
   END_RUNG
   // the same network as SCL:
   "DB7237_IDS_AND_PASSWORDS".ANY_ID_OK := NOT ("M_ONE" AND NOT "DB7237_IDS_AND_PASSWORDS".ID_OK[1] AND NOT "DB7237_IDS_AND_PASSWORDS".ID_OK[2] AND NOT "DB7237_IDS_AND_PASSWORDS".ID_OK[3] AND NOT "DB7237_IDS_AND_PASSWORDS".ID_OK[4] AND NOT "DB7237_IDS_AND_PASSWORDS".ID_OK[5]);
   "DB7237_IDS_AND_PASSWORDS".ANY_PASSWORD_OK := NOT ("M_ONE" AND NOT "DB7237_IDS_AND_PASSWORDS".ANY_PASSWORD_OK AND NOT "DB7237_IDS_AND_PASSWORDS".PASSWORD_OK[1] AND NOT "DB7237_IDS_AND_PASSWORDS".PASSWORD_OK[2] AND NOT "DB7237_IDS_AND_PASSWORDS".PASSWORD_OK[3] AND NOT "DB7237_IDS_AND_PASSWORDS".PASSWORD_OK[4] AND NOT "DB7237_IDS_AND_PASSWORDS".PASSWORD_OK[5]);
END_REGION

REGION Network 44: RESET PASSWORD
   RUNG wire#powerrail
      { S7_Templates := "SrcType := Byte" } NE_Contact(in1 := "LTLP_HMIProInterfaceData".noSoftKey, in2 := "DB7237_IDS_AND_PASSWORDS".SCREEN_ID_1)
      wire#w1
      Contact( "NETWORK_CHECK" )
      R_Coil( "DB7237_IDS_AND_PASSWORDS".RESET_PASSWORD )
   END_RUNG
   RUNG wire#powerrail
      { S7_Templates := "SrcType := Byte" } NE_Contact(in1 := "LTLP_HMIProInterfaceData".noFunctionKey, in2 := "DB7237_IDS_AND_PASSWORDS".SCREEN_ID_2)
   END_RUNG wire#w1
   // the same network as SCL:
   IF (("LTLP_HMIProInterfaceData".noSoftKey <> "DB7237_IDS_AND_PASSWORDS".SCREEN_ID_1) OR ("LTLP_HMIProInterfaceData".noFunctionKey <> "DB7237_IDS_AND_PASSWORDS".SCREEN_ID_2)) AND "NETWORK_CHECK" THEN
       "DB7237_IDS_AND_PASSWORDS".RESET_PASSWORD := FALSE;
   END_IF;
END_REGION

REGION Network 45: SCREEN LEVELS
   RUNG wire#powerrail
      Move(in := "LTLP_HMIProInterfaceData".noSoftKey, out1 => "DB7237_IDS_AND_PASSWORDS".SCREEN_ID_1)
      Move(in := "LTLP_HMIProInterfaceData".noFunctionKey, out1 => "DB7237_IDS_AND_PASSWORDS".SCREEN_ID_2)
   END_RUNG
   // the same network as SCL:
   "DB7237_IDS_AND_PASSWORDS".SCREEN_ID_1 := "LTLP_HMIProInterfaceData".noSoftKey;
   "DB7237_IDS_AND_PASSWORDS".SCREEN_ID_2 := "LTLP_HMIProInterfaceData".noFunctionKey;
END_REGION

REGION Network 46: RESET PASSWORD AUXILIARY
   RUNG wire#powerrail
      I_Contact( "DB7237_IDS_AND_PASSWORDS".RESET_PASSWORD )
      { S7_Templates := "time_type := Time" } "DB7237_IDS_AND_PASSWORDS".TIMER_RESET_PASSWORD_DELAY.TON(pt := "DB7237_IDS_AND_PASSWORDS".TIMER_RESET_PASSWORD_DELAY.PT, et =>)
      Coil( "DB7237_IDS_AND_PASSWORDS".RESET_PASSWORD_AUX )
   END_RUNG
   // the same network as SCL:
   "DB7237_IDS_AND_PASSWORDS".TIMER_RESET_PASSWORD_DELAY.TON(IN := NOT "DB7237_IDS_AND_PASSWORDS".RESET_PASSWORD,
                           PT := "DB7237_IDS_AND_PASSWORDS".TIMER_RESET_PASSWORD_DELAY.PT);
   "DB7237_IDS_AND_PASSWORDS".RESET_PASSWORD_AUX := "DB7237_IDS_AND_PASSWORDS".TIMER_RESET_PASSWORD_DELAY.Q;
END_REGION

REGION Network 47: TIMER RESET AUXILIARY
   RUNG wire#powerrail
      Contact( "DB7237_IDS_AND_PASSWORDS".ANY_ID_OK )
      Contact( "DB7237_IDS_AND_PASSWORDS".ANY_PASSWORD_OK )
      { S7_Templates := "time_type := Time" } "DB7237_IDS_AND_PASSWORDS".TIMER_RESET_PASSWORD.TON(pt := "DB7237_IDS_AND_PASSWORDS".TIMER_RESET_PASSWORD.PT, et =>)
      Coil( "DB7237_IDS_AND_PASSWORDS".AUX_TIMER_RESET )
   END_RUNG
   // the same network as SCL:
   "DB7237_IDS_AND_PASSWORDS".TIMER_RESET_PASSWORD.TON(IN := "DB7237_IDS_AND_PASSWORDS".ANY_ID_OK AND "DB7237_IDS_AND_PASSWORDS".ANY_PASSWORD_OK,
                           PT := "DB7237_IDS_AND_PASSWORDS".TIMER_RESET_PASSWORD.PT);
   "DB7237_IDS_AND_PASSWORDS".AUX_TIMER_RESET := "DB7237_IDS_AND_PASSWORDS".TIMER_RESET_PASSWORD.Q;
END_REGION

REGION Network 48: RESET ANY USER ID OK AND ANY PASSWORD OK
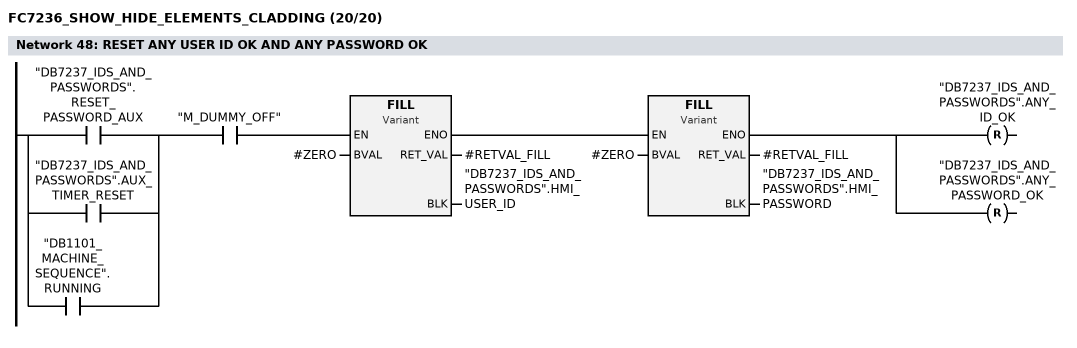
   RUNG wire#powerrail
      Contact( "DB7237_IDS_AND_PASSWORDS".RESET_PASSWORD_AUX )
      wire#w1
      Contact( "M_DUMMY_OFF" )
      { S7_Templates := "ptr_type := Variant" } FILL(BVAL := #ZERO, RET_VAL => #RETVAL_FILL, BLK => "DB7237_IDS_AND_PASSWORDS".HMI_USER_ID)
      { S7_Templates := "ptr_type := Variant" } FILL(BVAL := #ZERO, RET_VAL => #RETVAL_FILL, BLK => "DB7237_IDS_AND_PASSWORDS".HMI_PASSWORD)
      wire#w2
      R_Coil( "DB7237_IDS_AND_PASSWORDS".ANY_ID_OK )
   END_RUNG
   RUNG wire#powerrail
      Contact( "DB7237_IDS_AND_PASSWORDS".AUX_TIMER_RESET )
   END_RUNG wire#w1
   RUNG wire#powerrail
      Contact( "DB1101_MACHINE_SEQUENCE".RUNNING )
   END_RUNG wire#w1
   RUNG wire#w2
      R_Coil( "DB7237_IDS_AND_PASSWORDS".ANY_PASSWORD_OK )
   END_RUNG
   // the same network as SCL:
   #RETVAL_FILL := FILL(EN := ("DB7237_IDS_AND_PASSWORDS".RESET_PASSWORD_AUX OR "DB7237_IDS_AND_PASSWORDS".AUX_TIMER_RESET OR "DB1101_MACHINE_SEQUENCE".RUNNING) AND "M_DUMMY_OFF",
                        BVAL := #ZERO,
                        BLK => "DB7237_IDS_AND_PASSWORDS".HMI_USER_ID,
                        ENO => #_w1);
   #RETVAL_FILL := FILL(EN := #_w1, BVAL := #ZERO, BLK => "DB7237_IDS_AND_PASSWORDS".HMI_PASSWORD, ENO => #_w2);
   IF #_w2 THEN
       "DB7237_IDS_AND_PASSWORDS".ANY_ID_OK := FALSE;
       "DB7237_IDS_AND_PASSWORDS".ANY_PASSWORD_OK := FALSE;
   END_IF;
END_REGION
END_FUNCTION
